KUKA KRL program: EPS_2_25369_MH3A_A_20251128065458.src

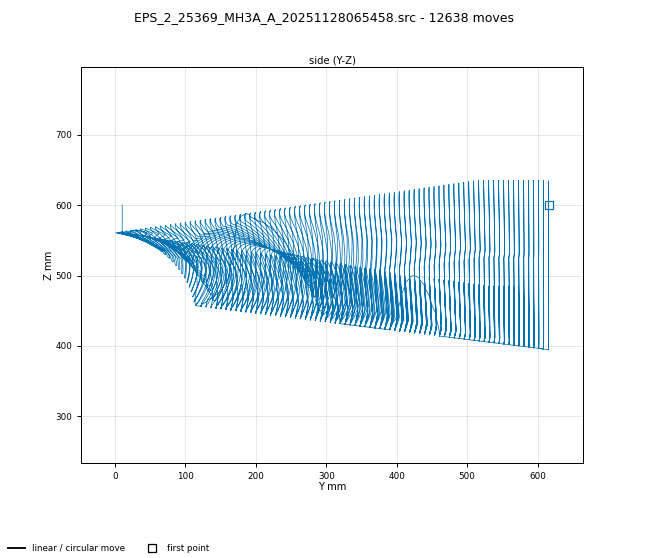
[picture p0: tool path of EPS_2_25369_MH3A_A_20251128065458.src, 12638 of 12640 moves have a stored position in this frame; points joined in program order, loops and branches not executed]
&ACCESS RVP
&REL 4
&COMMENT QRS 19112012
&PARAM EDITMASK = *
DEF PART()
EXT BAS (BAS_COMMAND :IN,REAL :IN )
INT I
BAS (#INITMOV,0 )

;KUKA QRS Post kuka4.cps  Date:22-06-2017 !

File_ID=2933

QRS_PRE_INIT()

;Init var - Until changes are made in qrs_pre_init
Outlet_Square_prg=0
Inlet_1_Square_prg=0
Inlet_2_Square_prg=0
Inlet_3_Square_prg=0
Inlet_4_Square_prg=0
Inlet_5_Square_prg=0

Outlet_1={X 0.000, Y 515.340, Z 534.500, B 0.000, E1 0.000 }
Inlet_1={X 0.000, Y 526.220, Z 384.500, B 0.000, E1 183.000 }
Inlet_2={X 0.000, Y 526.220, Z 384.500, B 0.000, E1 271.000 }
Outlet_1_type=201
Inlet_1_type=201
Inlet_2_type=201
;QRS#1=Sidecore dimensions
;QRS#2=200-8" PVC SDR 35
;QRS#3=200-8" PVC SDR 35
;QRS#4=200-8" PVC SDR 35
;QRS#5=
;QRS#6=
;QRS#7=
;QRS#8=
;QRS#9=12-08 PSX
;QRS#10=12-08 PSX
;QRS#11=12-08 PSX
;QRS#12=
;QRS#13=
;QRS#14=
;QRS#15=
;QRS#16=1220x127x914 3'
;QRS#17=EPS Height
;QRS#18=635
;QRS#19=*
;QRS#20= UPDATED VERSION 22-06-2017
;QRS#21=*
Outlet_Square=0100
Inlet_1_Square=0100
Inlet_2_Square=0100
Inlet_3_Square=0
Inlet_4_Square=0
Inlet_5_Square=0
Mill_Square=1
Outlet_Square_Prg=204
Inlet_1_Square_prg=204
Inlet_2_Square_prg=204

QRS_INIT()

$ADVANCE=5

; T1
PTP {E1 173.603,E2 173.603}
PTP {X 0,Y 615.513,A -85,B 0,C 180,E1 173.603,E2 173.603,E3 0,E4 0,E5 0,E6 0}
QRS_SPEED_INIT()
LIN {X 0,Y 615.513,Z 600,A -85,B 0,C 180,E1 173.603,E2 173.603,E3 0,E4 0,E5 0,E6 0} C_VEL
LIN {X 0,Y 615.513,Z 404.872,A -85,B 0,C 180,E1 173.603,E2 173.603} C_VEL
LIN {X 0,Y 615.513,Z 396.699,A -85,B 0,C 180,E1 173.603,E2 173.603} C_VEL
LIN {X 0,Y 615.495,Z 394.699,A -85,B 0,C 180,E1 173.416,E2 173.416} C_VEL
LIN {X 0,Y 615.488,Z 394.697,A -85,B 0,C 180,E1 170.801,E2 170.801} C_VEL
LIN {X 0,Y 615.484,Z 394.699,A -85,B 0,C 180,E1 168.139,E2 168.139} C_VEL
LIN {X 0,Y 615.49,Z 394.698,A -85,B 0,C 180,E1 165.451,E2 165.451} C_VEL
LIN {X 0,Y 615.49,Z 394.698,A -85,B 0,C 180,E1 162.729,E2 162.729} C_VEL
LIN {X 0,Y 615.486,Z 394.698,A -85,B 0,C 180,E1 159.967,E2 159.967} C_VEL
LIN {X 0,Y 615.489,Z 394.7,A -85,B 0,C 180,E1 157.155,E2 157.155} C_VEL
LIN {X 0,Y 615.486,Z 394.697,A -85,B 0,C 180,E1 154.432,E2 154.432} C_VEL
LIN {X 0,Y 615.493,Z 394.7,A -85,B 0,C 180,E1 151.549,E2 151.549} C_VEL
LIN {X 0,Y 615.483,Z 394.698,A -85,B 0,C 180,E1 148.915,E2 148.915} C_VEL
LIN {X 0,Y 615.486,Z 394.699,A -85,B 0,C 180,E1 146.466,E2 146.466} C_VEL
LIN {X 0,Y 615.491,Z 394.7,A -85,B 0,C 180,E1 144.166,E2 144.166} C_VEL
LIN {X 0,Y 615.493,Z 394.7,A -85,B 0,C 180,E1 141.931,E2 141.931} C_VEL
LIN {X 0,Y 615.48,Z 394.699,A -85,B 0,C 180,E1 139.393,E2 139.393} C_VEL
LIN {X 0,Y 615.498,Z 394.696,A -85,B 0,C 180,E1 136.756,E2 136.756} C_VEL
LIN {X 0,Y 615.493,Z 394.697,A -85,B 0,C 180,E1 133.998,E2 133.998} C_VEL
LIN {X 0,Y 615.49,Z 394.701,A -85,B 0,C 180,E1 131.094,E2 131.094} C_VEL
LIN {X 0,Y 615.493,Z 394.701,A -85,B 0,C 180,E1 128.904,E2 128.904} C_VEL
LIN {X 0,Y 615.483,Z 394.699,A -85,B 0,C 180,E1 126.425,E2 126.425} C_VEL
LIN {X 0,Y 615.488,Z 394.696,A -85,B 0,C 180,E1 124.022,E2 124.022} C_VEL
LIN {X 0,Y 615.493,Z 394.696,A -85,B 0,C 180,E1 121.685,E2 121.685} C_VEL
LIN {X 0,Y 615.488,Z 394.698,A -85,B 0,C 180,E1 119.406,E2 119.406} C_VEL
LIN {X 0,Y 615.491,Z 394.7,A -85,B 0,C 180,E1 117.045,E2 117.045} C_VEL
LIN {X 0,Y 615.479,Z 394.699,A -85,B 0,C 180,E1 114.272,E2 114.272} C_VEL
LIN {X 0,Y 615.49,Z 394.7,A -85,B 0,C 180,E1 111.432,E2 111.432} C_VEL
LIN {X 0,Y 615.482,Z 394.699,A -85,B 0,C 180,E1 108.602,E2 108.602} C_VEL
LIN {X 0,Y 615.492,Z 394.698,A -85,B 0,C 180,E1 105.905,E2 105.905} C_VEL
LIN {X 0,Y 615.48,Z 394.699,A -85,B 0,C 180,E1 103.201,E2 103.201} C_VEL
LIN {X 0,Y 615.487,Z 394.699,A -85,B 0,C 180,E1 100.527,E2 100.527} C_VEL
LIN {X 0,Y 615.492,Z 394.697,A -85,B 0,C 180,E1 98.247,E2 98.247} C_VEL
LIN {X 0,Y 615.49,Z 407.911,A -85,B 0,C 180,E1 97.793,E2 97.793} C_VEL
LIN {X 0,Y 615.49,Z 420.359,A -85,B 0,C 180,E1 97.216,E2 97.216} C_VEL
LIN {X 0,Y 615.488,Z 431.447,A -85,B 0,C 180,E1 96.557,E2 96.557} C_VEL
LIN {X 0,Y 615.498,Z 441.465,A -85,B 0,C 180,E1 95.816,E2 95.816} C_VEL
LIN {X 0,Y 615.498,Z 451.287,A -85,B 0,C 180,E1 94.913,E2 94.913} C_VEL
LIN {X 0,Y 615.497,Z 459.947,A -85,B 0,C 180,E1 93.928,E2 93.928} C_VEL
LIN {X 0,Y 615.497,Z 466.864,A -85,B 0,C 180,E1 92.945,E2 92.945} C_VEL
LIN {X 0,Y 615.5,Z 472.408,A -85,B 0,C 180,E1 91.963,E2 91.963} C_VEL
LIN {X 0,Y 615.497,Z 476.776,A -85,B 0,C 180,E1 90.981,E2 90.981} C_VEL
LIN {X 0,Y 615.496,Z 480.091,A -85,B 0,C 180,E1 90,E2 90} C_VEL
LIN {X 0,Y 615.498,Z 482.985,A -85,B 0,C 180,E1 88.691,E2 88.691} C_VEL
LIN {X 0,Y 615.499,Z 483.848,A -85,B 0,C 180,E1 88.037,E2 88.037} C_VEL
LIN {X 0,Y 615.496,Z 484.294,A -85,B 0,C 180,E1 87.382,E2 87.382} C_VEL
LIN {X 0,Y 615.495,Z 484.012,A -85,B 0,C 180,E1 86.071,E2 86.071} C_VEL
LIN {X 0,Y 615.495,Z 483.305,A -85,B 0,C 180,E1 85.415,E2 85.415} C_VEL
LIN {X 0,Y 615.496,Z 482.159,A -85,B 0,C 180,E1 84.759,E2 84.759} C_VEL
LIN {X 0,Y 615.497,Z 480.602,A -85,B 0,C 180,E1 84.101,E2 84.101} C_VEL
LIN {X 0,Y 615.497,Z 477.422,A -85,B 0,C 180,E1 83.102,E2 83.102} C_VEL
LIN {X 0,Y 615.495,Z 473.273,A -85,B 0,C 180,E1 82.124,E2 82.124} C_VEL
LIN {X 0,Y 615.496,Z 466.876,A -85,B 0,C 180,E1 80.967,E2 80.967} C_VEL
LIN {X 0,Y 615.497,Z 459.868,A -85,B 0,C 180,E1 79.972,E2 79.972} C_VEL
LIN {X 0,Y 615.498,Z 450.905,A -85,B 0,C 180,E1 78.958,E2 78.958} C_VEL
LIN {X 0,Y 615.497,Z 442.001,A -85,B 0,C 180,E1 78.139,E2 78.139} C_VEL
LIN {X 0,Y 615.484,Z 431.945,A -85,B 0,C 180,E1 77.386,E2 77.386} C_VEL
LIN {X 0,Y 615.477,Z 420.738,A -85,B 0,C 180,E1 76.714,E2 76.714} C_VEL
LIN {X 0,Y 615.487,Z 410.114,A -85,B 0,C 180,E1 76.21,E2 76.21} C_VEL
LIN {X 0,Y 615.492,Z 397.644,A -85,B 0,C 180,E1 75.758,E2 75.758} C_VEL
LIN {X 0,Y 615.493,Z 394.697,A -85,B 0,C 180,E1 75.662,E2 75.662} C_VEL
LIN {X 0,Y 615.487,Z 394.697,A -85,B 0,C 180,E1 73.413,E2 73.413} C_VEL
LIN {X 0,Y 615.475,Z 394.685,A -85,B 0,C 180,E1 70.661,E2 70.661} C_VEL
LIN {X 0,Y 615.493,Z 394.694,A -85,B 0,C 180,E1 67.864,E2 67.864} C_VEL
LIN {X 0,Y 615.488,Z 394.684,A -85,B 0,C 180,E1 65.008,E2 65.008} C_VEL
LIN {X 0,Y 615.48,Z 394.684,A -85,B 0,C 180,E1 62.822,E2 62.822} C_VEL
LIN {X 0,Y 615.497,Z 394.686,A -85,B 0,C 180,E1 60.205,E2 60.205} C_VEL
LIN {X 0,Y 615.479,Z 394.696,A -85,B 0,C 180,E1 57.542,E2 57.542} C_VEL
LIN {X 0,Y 615.499,Z 394.683,A -85,B 0,C 180,E1 55.185,E2 55.185} C_VEL
LIN {X 0,Y 615.477,Z 394.685,A -85,B 0,C 180,E1 52.757,E2 52.757} C_VEL
LIN {X 0,Y 615.498,Z 394.699,A -85,B 0,C 180,E1 49.91,E2 49.91} C_VEL
LIN {X 0,Y 615.481,Z 394.684,A -85,B 0,C 180,E1 46.954,E2 46.954} C_VEL
LIN {X 0,Y 615.49,Z 394.7,A -85,B 0,C 180,E1 43.997,E2 43.997} C_VEL
LIN {X 0,Y 615.485,Z 394.688,A -85,B 0,C 180,E1 41.474,E2 41.474} C_VEL
LIN {X 0,Y 615.478,Z 394.685,A -85,B 0,C 180,E1 38.905,E2 38.905} C_VEL
LIN {X 0,Y 615.488,Z 394.69,A -85,B 0,C 180,E1 36.425,E2 36.425} C_VEL
LIN {X 0,Y 615.484,Z 394.687,A -85,B 0,C 180,E1 33.533,E2 33.533} C_VEL
LIN {X 0,Y 615.478,Z 394.685,A -85,B 0,C 180,E1 30.921,E2 30.921} C_VEL
LIN {X 0,Y 615.491,Z 394.691,A -85,B 0,C 180,E1 28.45,E2 28.45} C_VEL
LIN {X 0,Y 615.486,Z 394.686,A -85,B 0,C 180,E1 25.568,E2 25.568} C_VEL
LIN {X 0,Y 615.475,Z 394.688,A -85,B 0,C 180,E1 22.845,E2 22.845} C_VEL
LIN {X 0,Y 615.487,Z 394.692,A -85,B 0,C 180,E1 20.556,E2 20.556} C_VEL
LIN {X 0,Y 615.482,Z 394.694,A -85,B 0,C 180,E1 17.957,E2 17.957} C_VEL
LIN {X 0,Y 615.486,Z 394.683,A -85,B 0,C 180,E1 15.226,E2 15.226} C_VEL
LIN {X 0,Y 615.486,Z 394.696,A -85,B 0,C 180,E1 12.53,E2 12.53} C_VEL
LIN {X 0,Y 615.483,Z 394.699,A -85,B 0,C 180,E1 10.236,E2 10.236} C_VEL
LIN {X 0,Y 615.478,Z 407.188,A -85,B 0,C 180,E1 9.821,E2 9.821} C_VEL
LIN {X 0,Y 615.486,Z 419.115,A -85,B 0,C 180,E1 9.282,E2 9.282} C_VEL
LIN {X 0,Y 615.487,Z 430.482,A -85,B 0,C 180,E1 8.619,E2 8.619} C_VEL
LIN {X 0,Y 615.498,Z 440.718,A -85,B 0,C 180,E1 7.876,E2 7.876} C_VEL
LIN {X 0,Y 615.499,Z 449.87,A -85,B 0,C 180,E1 7.057,E2 7.057} C_VEL
LIN {X 0,Y 615.496,Z 458.846,A -85,B 0,C 180,E1 6.063,E2 6.063} C_VEL
LIN {X 0,Y 615.497,Z 466.028,A -85,B 0,C 180,E1 5.077,E2 5.077} C_VEL
LIN {X 0,Y 615.496,Z 470.874,A -85,B 0,C 180,E1 4.257,E2 4.257} C_VEL
LIN {X 0,Y 615.496,Z 475.586,A -85,B 0,C 180,E1 3.273,E2 3.273} C_VEL
LIN {X 0,Y 615.498,Z 479.197,A -85,B 0,C 180,E1 2.291,E2 2.291} C_VEL
LIN {X 0,Y 615.496,Z 481.817,A -85,B 0,C 180,E1 1.309,E2 1.309} C_VEL
LIN {X 0,Y 615.495,Z 483.889,A -85,B 0,C 180,E1 0,E2 0} C_VEL
LIN {X 0,Y 615.496,Z 484.331,A -85,B 0,C 180,E1 -1.308,E2 -1.308} C_VEL
LIN {X 0,Y 615.495,Z 483.257,A -85,B 0,C 180,E1 -2.618,E2 -2.618} C_VEL
LIN {X 0,Y 615.497,Z 482.09,A -85,B 0,C 180,E1 -3.273,E2 -3.273} C_VEL
LIN {X 0,Y 615.494,Z 480.523,A -85,B 0,C 180,E1 -3.928,E2 -3.928} C_VEL
LIN {X 0,Y 615.494,Z 477.369,A -85,B 0,C 180,E1 -4.913,E2 -4.913} C_VEL
LIN {X 0,Y 615.498,Z 473.162,A -85,B 0,C 180,E1 -5.898,E2 -5.898} C_VEL
LIN {X 0,Y 615.497,Z 466.732,A -85,B 0,C 180,E1 -7.057,E2 -7.057} C_VEL
LIN {X 0,Y 615.498,Z 459.768,A -85,B 0,C 180,E1 -8.041,E2 -8.041} C_VEL
LIN {X 0,Y 615.497,Z 450.99,A -85,B 0,C 180,E1 -9.033,E2 -9.033} C_VEL
LIN {X 0,Y 615.499,Z 441.987,A -85,B 0,C 180,E1 -9.862,E2 -9.862} C_VEL
LIN {X 0,Y 615.488,Z 431.924,A -85,B 0,C 180,E1 -10.615,E2 -10.615} C_VEL
LIN {X 0,Y 615.488,Z 420.906,A -85,B 0,C 180,E1 -11.276,E2 -11.276} C_VEL
LIN {X 0,Y 615.487,Z 408.448,A -85,B 0,C 180,E1 -11.861,E2 -11.861} C_VEL
LIN {X 0,Y 615.489,Z 396.407,A -85,B 0,C 180,E1 -12.279,E2 -12.279} C_VEL
LIN {X 0,Y 615.488,Z 394.694,A -85,B 0,C 180,E1 -12.342,E2 -12.342} C_VEL
LIN {X 0,Y 615.49,Z 394.692,A -85,B 0,C 180,E1 -15.226,E2 -15.226} C_VEL
LIN {X 0,Y 615.477,Z 394.696,A -85,B 0,C 180,E1 -17.957,E2 -17.957} C_VEL
LIN {X 0,Y 615.477,Z 394.696,A -85,B 0,C 180,E1 -20.731,E2 -20.731} C_VEL
LIN {X 0,Y 615.486,Z 394.694,A -85,B 0,C 180,E1 -23.556,E2 -23.556} C_VEL
LIN {X 0,Y 615.493,Z 394.691,A -85,B 0,C 180,E1 -26.444,E2 -26.444} C_VEL
LIN {X 0,Y 615.492,Z 394.692,A -85,B 0,C 180,E1 -29.406,E2 -29.406} C_VEL
LIN {X 0,Y 615.492,Z 394.693,A -85,B 0,C 180,E1 -32.331,E2 -32.331} C_VEL
LIN {X 0,Y 615.477,Z 394.695,A -85,B 0,C 180,E1 -34.816,E2 -34.816} C_VEL
LIN {X 0,Y 615.494,Z 394.694,A -85,B 0,C 180,E1 -37.242,E2 -37.242} C_VEL
LIN {X 0,Y 615.488,Z 394.695,A -85,B 0,C 180,E1 -40.089,E2 -40.089} C_VEL
LIN {X 0,Y 615.499,Z 394.696,A -85,B 0,C 180,E1 -42.352,E2 -42.352} C_VEL
LIN {X 0,Y 615.48,Z 394.699,A -85,B 0,C 180,E1 -45.069,E2 -45.069} C_VEL
LIN {X 0,Y 615.487,Z 394.699,A -85,B 0,C 180,E1 -47.92,E2 -47.92} C_VEL
LIN {X 0,Y 615.494,Z 394.691,A -85,B 0,C 180,E1 -50.25,E2 -50.25} C_VEL
LIN {X 0,Y 615.482,Z 394.694,A -85,B 0,C 180,E1 -53.064,E2 -53.064} C_VEL
LIN {X 0,Y 615.479,Z 394.815,A -85,B 0,C 180,E1 -54.534,E2 -54.534} C_VEL
LIN {X 0,Y 615.489,Z 408.626,A -85,B 0,C 180,E1 -57.154,E2 -57.154} C_VEL
LIN {X 0,Y 615.476,Z 422.321,A -85,B 0,C 180,E1 -59.839,E2 -59.839} C_VEL
LIN {X 0,Y 615.481,Z 436.016,A -85,B 0,C 180,E1 -62.454,E2 -62.454} C_VEL
LIN {X 0,Y 615.497,Z 449.705,A -85,B 0,C 180,E1 -65.008,E2 -65.008} C_VEL
LIN {X 0,Y 615.487,Z 465.337,A -85,B 0,C 180,E1 -67.863,E2 -67.863} C_VEL
LIN {X 0,Y 615.492,Z 480.953,A -85,B 0,C 180,E1 -70.662,E2 -70.662} C_VEL
LIN {X 0,Y 615.492,Z 496.555,A -85,B 0,C 180,E1 -73.413,E2 -73.413} C_VEL
LIN {X 0,Y 615.498,Z 512.141,A -85,B 0,C 180,E1 -76.126,E2 -76.126} C_VEL
LIN {X 0,Y 615.482,Z 524.926,A -85,B 0,C 180,E1 -78.327,E2 -78.327} C_VEL
LIN {X 0,Y 615.477,Z 538.234,A -85,B 0,C 180,E1 -78.556,E2 -78.556} C_VEL
LIN {X 0,Y 615.489,Z 551.332,A -85,B 0,C 180,E1 -78.922,E2 -78.922} C_VEL
LIN {X 0,Y 615.48,Z 563.127,A -85,B 0,C 180,E1 -79.383,E2 -79.383} C_VEL
LIN {X 0,Y 615.486,Z 574.572,A -85,B 0,C 180,E1 -79.972,E2 -79.972} C_VEL
LIN {X 0,Y 615.499,Z 586.019,A -85,B 0,C 180,E1 -80.718,E2 -80.718} C_VEL
LIN {X 0,Y 615.498,Z 595.255,A -85,B 0,C 180,E1 -81.463,E2 -81.463} C_VEL
LIN {X 0,Y 615.499,Z 603.652,A -85,B 0,C 180,E1 -82.289,E2 -82.289} C_VEL
LIN {X 0,Y 615.497,Z 611.69,A -85,B 0,C 180,E1 -83.259,E2 -83.259} C_VEL
LIN {X 0,Y 615.498,Z 617.422,A -85,B 0,C 180,E1 -84.101,E2 -84.101} C_VEL
LIN {X 0,Y 615.497,Z 622.871,A -85,B 0,C 180,E1 -85.087,E2 -85.087} C_VEL
LIN {X 0,Y 615.496,Z 627.14,A -85,B 0,C 180,E1 -86.071,E2 -86.071} C_VEL
LIN {X 0,Y 615.495,Z 629.398,A -85,B 0,C 180,E1 -86.727,E2 -86.727} C_VEL
LIN {X 0,Y 615.497,Z 631.232,A -85,B 0,C 180,E1 -87.382,E2 -87.382} C_VEL
LIN {X 0,Y 615.497,Z 632.608,A -85,B 0,C 180,E1 -88.037,E2 -88.037} C_VEL
LIN {X 0,Y 615.496,Z 634.173,A -85,B 0,C 180,E1 -89.346,E2 -89.346} C_VEL
LIN {X 0,Y 615.494,Z 634.389,A -85,B 0,C 180,E1 -90,E2 -90} C_VEL
LIN {X 0,Y 615.496,Z 633.58,A -85,B 0,C 180,E1 -91.308,E2 -91.308} C_VEL
LIN {X 0,Y 615.497,Z 632.608,A -85,B 0,C 180,E1 -91.963,E2 -91.963} C_VEL
LIN {X 0,Y 615.497,Z 631.233,A -85,B 0,C 180,E1 -92.618,E2 -92.618} C_VEL
LIN {X 0,Y 615.496,Z 628.35,A -85,B 0,C 180,E1 -93.6,E2 -93.6} C_VEL
LIN {X 0,Y 615.498,Z 624.442,A -85,B 0,C 180,E1 -94.584,E2 -94.584} C_VEL
LIN {X 0,Y 615.499,Z 619.405,A -85,B 0,C 180,E1 -95.57,E2 -95.57} C_VEL
LIN {X 0,Y 615.497,Z 612.869,A -85,B 0,C 180,E1 -96.583,E2 -96.583} C_VEL
LIN {X 0,Y 615.497,Z 605.134,A -85,B 0,C 180,E1 -97.545,E2 -97.545} C_VEL
LIN {X 0,Y 615.498,Z 597.046,A -85,B 0,C 180,E1 -98.371,E2 -98.371} C_VEL
LIN {X 0,Y 615.499,Z 587.169,A -85,B 0,C 180,E1 -99.198,E2 -99.198} C_VEL
LIN {X 0,Y 615.488,Z 575.983,A -85,B 0,C 180,E1 -99.945,E2 -99.945} C_VEL
LIN {X 0,Y 615.478,Z 565.026,A -85,B 0,C 180,E1 -100.527,E2 -100.527} C_VEL
LIN {X 0,Y 615.489,Z 552.505,A -85,B 0,C 180,E1 -101.039,E2 -101.039} C_VEL
LIN {X 0,Y 615.477,Z 540.071,A -85,B 0,C 180,E1 -101.402,E2 -101.402} C_VEL
LIN {X 0,Y 615.481,Z 526.474,A -85,B 0,C 180,E1 -101.652,E2 -101.652} C_VEL
LIN {X 0,Y 615.483,Z 524.799,A -85,B 0,C 180,E1 -101.694,E2 -101.694} C_VEL
LIN {X 0,Y 615.48,Z 510.017,A -85,B 0,C 180,E1 -104.242,E2 -104.242} C_VEL
LIN {X 0,Y 615.494,Z 494.605,A -85,B 0,C 180,E1 -106.928,E2 -106.928} C_VEL
LIN {X 0,Y 615.495,Z 479.002,A -85,B 0,C 180,E1 -109.685,E2 -109.685} C_VEL
LIN {X 0,Y 615.494,Z 462.802,A -85,B 0,C 180,E1 -112.595,E2 -112.595} C_VEL
LIN {X 0,Y 615.485,Z 448.151,A -85,B 0,C 180,E1 -115.279,E2 -115.279} C_VEL
LIN {X 0,Y 615.493,Z 434.061,A -85,B 0,C 180,E1 -117.915,E2 -117.915} C_VEL
LIN {X 0,Y 615.478,Z 420.366,A -85,B 0,C 180,E1 -120.54,E2 -120.54} C_VEL
LIN {X 0,Y 615.491,Z 406.665,A -85,B 0,C 180,E1 -123.236,E2 -123.236} C_VEL
LIN {X 0,Y 615.482,Z 394.698,A -85,B 0,C 180,E1 -125.516,E2 -125.516} C_VEL
LIN {X 0,Y 615.493,Z 394.699,A -85,B 0,C 180,E1 -128.068,E2 -128.068} C_VEL
LIN {X 0,Y 615.493,Z 394.697,A -85,B 0,C 180,E1 -130.606,E2 -130.606} C_VEL
LIN {X 0,Y 615.481,Z 394.699,A -85,B 0,C 180,E1 -133.245,E2 -133.245} C_VEL
LIN {X 0,Y 615.485,Z 394.7,A -85,B 0,C 180,E1 -136.003,E2 -136.003} C_VEL
LIN {X 0,Y 615.496,Z 394.698,A -85,B 0,C 180,E1 -138.905,E2 -138.905} C_VEL
LIN {X 0,Y 615.493,Z 394.699,A -85,B 0,C 180,E1 -141.096,E2 -141.096} C_VEL
LIN {X 0,Y 615.495,Z 394.697,A -85,B 0,C 180,E1 -143.576,E2 -143.576} C_VEL
LIN {X 0,Y 615.486,Z 394.7,A -85,B 0,C 180,E1 -146.466,E2 -146.466} C_VEL
LIN {X 0,Y 615.481,Z 394.7,A -85,B 0,C 180,E1 -149.08,E2 -149.08} C_VEL
LIN {X 0,Y 615.492,Z 394.696,A -85,B 0,C 180,E1 -151.549,E2 -151.549} C_VEL
LIN {X 0,Y 615.496,Z 394.697,A -85,B 0,C 180,E1 -154.43,E2 -154.43} C_VEL
LIN {X 0,Y 615.485,Z 394.698,A -85,B 0,C 180,E1 -157.155,E2 -157.155} C_VEL
LIN {X 0,Y 615.487,Z 394.7,A -85,B 0,C 180,E1 -159.444,E2 -159.444} C_VEL
LIN {X 0,Y 615.483,Z 394.699,A -85,B 0,C 180,E1 -162.043,E2 -162.043} C_VEL
LIN {X 0,Y 615.495,Z 394.696,A -85,B 0,C 180,E1 -164.774,E2 -164.774} C_VEL
LIN {X 0,Y 615.493,Z 394.697,A -85,B 0,C 180,E1 -167.47,E2 -167.47} C_VEL
LIN {X 0,Y 615.479,Z 394.7,A -85,B 0,C 180,E1 -170.138,E2 -170.138} C_VEL
LIN {X 0,Y 615.484,Z 394.701,A -85,B 0,C 180,E1 -172.784,E2 -172.784} C_VEL
LIN {X 0,Y 615.492,Z 394.696,A -85,B 0,C 180,E1 -175.416,E2 -175.416} C_VEL
LIN {X 0,Y 615.5,Z 394.7,A -85,B 0,C 180,E1 -178.037,E2 -178.037} C_VEL
LIN {X 0,Y 615.489,Z 394.696,A -85,B 0,C 180,E1 -180.654,E2 -180.654} C_VEL
LIN {X 0,Y 615.486,Z 394.7,A -85,B 0,C 180,E1 -183.273,E2 -183.273} C_VEL
LIN {X 0,Y 615.482,Z 394.699,A -85,B 0,C 180,E1 -185.899,E2 -185.899} C_VEL
LIN {X 0,Y 615.495,Z 394.699,A -85,B 0,C 180,E1 -186.584,E2 -186.584} C_VEL
LIN {X 0,Y 614.812,Z 394.843,A -85,B 0,C 180,E1 -187.13,E2 -187.13} C_VEL
LIN {X 0,Y 611.974,Z 395.258,A -85,B 0,C 180,E1 -188.016,E2 -188.016} C_VEL
LIN {X 0,Y 609.584,Z 395.566,A -85,B 0,C 180,E1 -188.728,E2 -188.728} C_VEL
LIN {X 0,Y 608.551,Z 395.684,A -85,B 0,C 180,E1 -189.278,E2 -189.278} C_VEL
LIN {X 0,Y 608.462,Z 395.694,A -85,B 0,C 180,E1 -189.464,E2 -189.464} C_VEL
LIN {X 0,Y 608.462,Z 395.696,A -85,B 0,C 180,E1 -192,E2 -192} C_VEL
LIN {X 0,Y 608.478,Z 395.692,A -85,B 0,C 180,E1 -194.721,E2 -194.721} C_VEL
LIN {X 0,Y 608.454,Z 395.697,A -85,B 0,C 180,E1 -197.477,E2 -197.477} C_VEL
LIN {X 0,Y 608.467,Z 395.693,A -85,B 0,C 180,E1 -200.274,E2 -200.274} C_VEL
LIN {X 0,Y 608.461,Z 395.694,A -85,B 0,C 180,E1 -202.477,E2 -202.477} C_VEL
LIN {X 0,Y 608.461,Z 395.694,A -85,B 0,C 180,E1 -204.571,E2 -204.571} C_VEL
LIN {X 0,Y 608.48,Z 395.694,A -85,B 0,C 180,E1 -207.207,E2 -207.207} C_VEL
LIN {X 0,Y 608.466,Z 395.693,A -85,B 0,C 180,E1 -209.971,E2 -209.971} C_VEL
LIN {X 0,Y 608.463,Z 395.695,A -85,B 0,C 180,E1 -212.879,E2 -212.879} C_VEL
LIN {X 0,Y 608.444,Z 395.696,A -85,B 0,C 180,E1 -215.278,E2 -215.278} C_VEL
LIN {X 0,Y 608.473,Z 395.693,A -85,B 0,C 180,E1 -217.746,E2 -217.746} C_VEL
LIN {X 0,Y 608.448,Z 395.698,A -85,B 0,C 180,E1 -220.329,E2 -220.329} C_VEL
LIN {X 0,Y 608.485,Z 395.692,A -85,B 0,C 180,E1 -223.31,E2 -223.31} C_VEL
LIN {X 0,Y 608.478,Z 395.692,A -85,B 0,C 180,E1 -226.131,E2 -226.131} C_VEL
LIN {X 0,Y 608.459,Z 395.696,A -85,B 0,C 180,E1 -228.824,E2 -228.824} C_VEL
LIN {X 0,Y 608.472,Z 395.693,A -85,B 0,C 180,E1 -231.412,E2 -231.412} C_VEL
LIN {X 0,Y 608.465,Z 395.694,A -85,B 0,C 180,E1 -233.953,E2 -233.953} C_VEL
LIN {X 0,Y 608.472,Z 395.694,A -85,B 0,C 180,E1 -236.33,E2 -236.33} C_VEL
LIN {X 0,Y 608.483,Z 395.694,A -85,B 0,C 180,E1 -238.728,E2 -238.728} C_VEL
LIN {X 0,Y 608.471,Z 395.693,A -85,B 0,C 180,E1 -241.381,E2 -241.381} C_VEL
LIN {X 0,Y 608.443,Z 395.698,A -85,B 0,C 180,E1 -243.964,E2 -243.964} C_VEL
LIN {X 0,Y 608.468,Z 395.695,A -85,B 0,C 180,E1 -246.155,E2 -246.155} C_VEL
LIN {X 0,Y 608.471,Z 395.695,A -85,B 0,C 180,E1 -248.309,E2 -248.309} C_VEL
LIN {X 0,Y 608.457,Z 395.694,A -85,B 0,C 180,E1 -251.131,E2 -251.131} C_VEL
LIN {X 0,Y 608.463,Z 395.697,A -85,B 0,C 180,E1 -253.906,E2 -253.906} C_VEL
LIN {X 0,Y 608.462,Z 395.694,A -85,B 0,C 180,E1 -256.644,E2 -256.644} C_VEL
LIN {X 0,Y 608.467,Z 395.696,A -85,B 0,C 180,E1 -259.35,E2 -259.35} C_VEL
LIN {X 0,Y 608.464,Z 395.712,A -85,B 0,C 180,E1 -261.657,E2 -261.657} C_VEL
LIN {X 0,Y 608.521,Z 407.891,A -85,B 0,C 180,E1 -262.076,E2 -262.076} C_VEL
LIN {X 0,Y 608.507,Z 419.64,A -85,B 0,C 180,E1 -262.618,E2 -262.618} C_VEL
LIN {X 0,Y 608.48,Z 430.93,A -85,B 0,C 180,E1 -263.284,E2 -263.284} C_VEL
LIN {X 0,Y 608.498,Z 441.131,A -85,B 0,C 180,E1 -264.034,E2 -264.034} C_VEL
LIN {X 0,Y 608.483,Z 450.335,A -85,B 0,C 180,E1 -264.865,E2 -264.865} C_VEL
LIN {X 0,Y 608.474,Z 459.266,A -85,B 0,C 180,E1 -265.86,E2 -265.86} C_VEL
LIN {X 0,Y 608.459,Z 466.478,A -85,B 0,C 180,E1 -266.855,E2 -266.855} C_VEL
LIN {X 0,Y 608.46,Z 471.352,A -85,B 0,C 180,E1 -267.683,E2 -267.683} C_VEL
LIN {X 0,Y 608.449,Z 476.1,A -85,B 0,C 180,E1 -268.676,E2 -268.676} C_VEL
LIN {X 0,Y 608.441,Z 479.749,A -85,B 0,C 180,E1 -269.669,E2 -269.669} C_VEL
LIN {X 0,Y 608.437,Z 482.397,A -85,B 0,C 180,E1 -270.662,E2 -270.662} C_VEL
LIN {X 0,Y 608.45,Z 483.641,A -85,B 0,C 180,E1 -271.324,E2 -271.324} C_VEL
LIN {X 0,Y 608.444,Z 484.493,A -85,B 0,C 180,E1 -271.986,E2 -271.986} C_VEL
LIN {X 0,Y 608.422,Z 484.944,A -85,B 0,C 180,E1 -273.311,E2 -273.311} C_VEL
LIN {X 0,Y 608.432,Z 484.595,A -85,B 0,C 180,E1 -273.974,E2 -273.974} C_VEL
LIN {X 0,Y 608.428,Z 483.852,A -85,B 0,C 180,E1 -274.638,E2 -274.638} C_VEL
LIN {X 0,Y 608.438,Z 482.668,A -85,B 0,C 180,E1 -275.302,E2 -275.302} C_VEL
LIN {X 0,Y 608.448,Z 479.169,A -85,B 0,C 180,E1 -276.603,E2 -276.603} C_VEL
LIN {X 0,Y 608.449,Z 475.161,A -85,B 0,C 180,E1 -277.633,E2 -277.633} C_VEL
LIN {X 0,Y 608.451,Z 470.1,A -85,B 0,C 180,E1 -278.636,E2 -278.636} C_VEL
LIN {X 0,Y 608.467,Z 463.732,A -85,B 0,C 180,E1 -279.642,E2 -279.642} C_VEL
LIN {X 0,Y 608.451,Z 455.728,A -85,B 0,C 180,E1 -280.65,E2 -280.65} C_VEL
LIN {X 0,Y 608.471,Z 447.556,A -85,B 0,C 180,E1 -281.493,E2 -281.493} C_VEL
LIN {X 0,Y 608.477,Z 437.568,A -85,B 0,C 180,E1 -282.338,E2 -282.338} C_VEL
LIN {X 0,Y 608.498,Z 426.247,A -85,B 0,C 180,E1 -283.101,E2 -283.101} C_VEL
LIN {X 0,Y 608.503,Z 415.135,A -85,B 0,C 180,E1 -283.696,E2 -283.696} C_VEL
LIN {X 0,Y 608.533,Z 402.778,A -85,B 0,C 180,E1 -284.207,E2 -284.207} C_VEL
LIN {X 0,Y 608.466,Z 395.697,A -85,B 0,C 180,E1 -284.443,E2 -284.443} C_VEL
LIN {X 0,Y 608.446,Z 395.693,A -85,B 0,C 180,E1 -286.784,E2 -286.784} C_VEL
LIN {X 0,Y 608.449,Z 395.688,A -85,B 0,C 180,E1 -289.571,E2 -289.571} C_VEL
LIN {X 0,Y 608.465,Z 395.694,A -85,B 0,C 180,E1 -292.476,E2 -292.476} C_VEL
LIN {X 0,Y 608.457,Z 395.693,A -85,B 0,C 180,E1 -294.571,E2 -294.571} C_VEL
LIN {X 0,Y 608.477,Z 395.684,A -85,B 0,C 180,E1 -297.206,E2 -297.206} C_VEL
LIN {X 0,Y 608.477,Z 395.69,A -85,B 0,C 180,E1 -299.972,E2 -299.972} C_VEL
LIN {X 0,Y 608.452,Z 395.689,A -85,B 0,C 180,E1 -302.88,E2 -302.88} C_VEL
LIN {X 0,Y 608.447,Z 395.688,A -85,B 0,C 180,E1 -305.278,E2 -305.278} C_VEL
LIN {X 0,Y 608.477,Z 395.694,A -85,B 0,C 180,E1 -308.241,E2 -308.241} C_VEL
LIN {X 0,Y 608.457,Z 395.687,A -85,B 0,C 180,E1 -311.341,E2 -311.341} C_VEL
LIN {X 0,Y 608.459,Z 395.694,A -85,B 0,C 180,E1 -314.264,E2 -314.264} C_VEL
LIN {X 0,Y 608.453,Z 395.687,A -85,B 0,C 180,E1 -317.04,E2 -317.04} C_VEL
LIN {X 0,Y 608.458,Z 395.692,A -85,B 0,C 180,E1 -319.697,E2 -319.697} C_VEL
LIN {X 0,Y 608.472,Z 395.691,A -85,B 0,C 180,E1 -322.254,E2 -322.254} C_VEL
LIN {X 0,Y 608.444,Z 395.689,A -85,B 0,C 180,E1 -325.096,E2 -325.096} C_VEL
LIN {X 0,Y 608.461,Z 395.69,A -85,B 0,C 180,E1 -327.478,E2 -327.478} C_VEL
LIN {X 0,Y 608.463,Z 395.691,A -85,B 0,C 180,E1 -330.22,E2 -330.22} C_VEL
LIN {X 0,Y 608.478,Z 395.684,A -85,B 0,C 180,E1 -332.794,E2 -332.794} C_VEL
LIN {X 0,Y 608.454,Z 395.691,A -85,B 0,C 180,E1 -335.429,E2 -335.429} C_VEL
LIN {X 0,Y 608.472,Z 395.687,A -85,B 0,C 180,E1 -338.308,E2 -338.308} C_VEL
LIN {X 0,Y 608.472,Z 395.688,A -85,B 0,C 180,E1 -341.285,E2 -341.285} C_VEL
LIN {X 0,Y 608.458,Z 395.694,A -85,B 0,C 180,E1 -343.906,E2 -343.906} C_VEL
LIN {X 0,Y 608.461,Z 395.686,A -85,B 0,C 180,E1 -346.643,E2 -346.643} C_VEL
LIN {X 0,Y 608.477,Z 395.695,A -85,B 0,C 180,E1 -349.645,E2 -349.645} C_VEL
LIN {X 0,Y 608.51,Z 408.661,A -85,B 0,C 180,E1 -350.107,E2 -350.107} C_VEL
LIN {X 0,Y 608.503,Z 421.068,A -85,B 0,C 180,E1 -350.695,E2 -350.695} C_VEL
LIN {X 0,Y 608.501,Z 432.147,A -85,B 0,C 180,E1 -351.364,E2 -351.364} C_VEL
LIN {X 0,Y 608.494,Z 441.129,A -85,B 0,C 180,E1 -352.033,E2 -352.033} C_VEL
LIN {X 0,Y 608.467,Z 450.36,A -85,B 0,C 180,E1 -352.867,E2 -352.867} C_VEL
LIN {X 0,Y 608.446,Z 459.315,A -85,B 0,C 180,E1 -353.866,E2 -353.866} C_VEL
LIN {X 0,Y 608.446,Z 466.538,A -85,B 0,C 180,E1 -354.864,E2 -354.864} C_VEL
LIN {X 0,Y 608.441,Z 471.413,A -85,B 0,C 180,E1 -355.694,E2 -355.694} C_VEL
LIN {X 0,Y 608.43,Z 476.157,A -85,B 0,C 180,E1 -356.689,E2 -356.689} C_VEL
LIN {X 0,Y 608.43,Z 479.793,A -85,B 0,C 180,E1 -357.683,E2 -357.683} C_VEL
LIN {X 0,Y 608.448,Z 482.428,A -85,B 0,C 180,E1 -358.676,E2 -358.676} C_VEL
LIN {X 0,Y 608.436,Z 484.505,A -85,B 0,C 180,E1 -360,E2 -360} C_VEL
LIN {X 0,Y 608.448,Z 484.941,A -85,B 0,C 180,E1 -361.324,E2 -361.324} C_VEL
LIN {X 0,Y 608.442,Z 484.587,A -85,B 0,C 180,E1 -361.986,E2 -361.986} C_VEL
LIN {X 0,Y 608.422,Z 483.836,A -85,B 0,C 180,E1 -362.648,E2 -362.648} C_VEL
LIN {X 0,Y 608.425,Z 482.651,A -85,B 0,C 180,E1 -363.311,E2 -363.311} C_VEL
LIN {X 0,Y 608.432,Z 480.116,A -85,B 0,C 180,E1 -364.306,E2 -364.306} C_VEL
LIN {X 0,Y 608.441,Z 476.58,A -85,B 0,C 180,E1 -365.302,E2 -365.302} C_VEL
LIN {X 0,Y 608.452,Z 471.56,A -85,B 0,C 180,E1 -366.369,E2 -366.369} C_VEL
LIN {X 0,Y 608.451,Z 464.92,A -85,B 0,C 180,E1 -367.466,E2 -367.466} C_VEL
LIN {X 0,Y 608.464,Z 457.315,A -85,B 0,C 180,E1 -368.469,E2 -368.469} C_VEL
LIN {X 0,Y 608.46,Z 449.539,A -85,B 0,C 180,E1 -369.306,E2 -369.306} C_VEL
LIN {X 0,Y 608.491,Z 438.955,A -85,B 0,C 180,E1 -370.229,E2 -370.229} C_VEL
LIN {X 0,Y 608.494,Z 428.487,A -85,B 0,C 180,E1 -370.966,E2 -370.966} C_VEL
LIN {X 0,Y 608.506,Z 417.621,A -85,B 0,C 180,E1 -371.576,E2 -371.576} C_VEL
LIN {X 0,Y 608.519,Z 404.962,A -85,B 0,C 180,E1 -372.125,E2 -372.125} C_VEL
LIN {X 0,Y 608.471,Z 395.691,A -85,B 0,C 180,E1 -372.444,E2 -372.444} C_VEL
LIN {X 0,Y 608.476,Z 395.69,A -85,B 0,C 180,E1 -375.406,E2 -375.406} C_VEL
LIN {X 0,Y 608.443,Z 395.694,A -85,B 0,C 180,E1 -378.172,E2 -378.172} C_VEL
LIN {X 0,Y 608.457,Z 395.693,A -85,B 0,C 180,E1 -380.982,E2 -380.982} C_VEL
LIN {X 0,Y 608.449,Z 395.697,A -85,B 0,C 180,E1 -383.124,E2 -383.124} C_VEL
LIN {X 0,Y 608.481,Z 395.694,A -85,B 0,C 180,E1 -385.722,E2 -385.722} C_VEL
LIN {X 0,Y 608.48,Z 395.694,A -85,B 0,C 180,E1 -388.62,E2 -388.62} C_VEL
LIN {X 0,Y 608.448,Z 395.698,A -85,B 0,C 180,E1 -391.318,E2 -391.318} C_VEL
LIN {X 0,Y 608.475,Z 395.691,A -85,B 0,C 180,E1 -393.735,E2 -393.735} C_VEL
LIN {X 0,Y 608.449,Z 395.694,A -85,B 0,C 180,E1 -396.092,E2 -396.092} C_VEL
LIN {X 0,Y 608.436,Z 395.697,A -85,B 0,C 180,E1 -398.591,E2 -398.591} C_VEL
LIN {X 0,Y 608.462,Z 395.694,A -85,B 0,C 180,E1 -401.342,E2 -401.342} C_VEL
LIN {X 0,Y 608.464,Z 395.693,A -85,B 0,C 180,E1 -404.264,E2 -404.264} C_VEL
LIN {X 0,Y 608.455,Z 395.694,A -85,B 0,C 180,E1 -407.04,E2 -407.04} C_VEL
LIN {X 0,Y 608.456,Z 395.695,A -85,B 0,C 180,E1 -409.697,E2 -409.697} C_VEL
LIN {X 0,Y 608.467,Z 395.697,A -85,B 0,C 180,E1 -412.253,E2 -412.253} C_VEL
LIN {X 0,Y 608.485,Z 395.82,A -85,B 0,C 180,E1 -414.369,E2 -414.369} C_VEL
LIN {X 0,Y 608.571,Z 407.184,A -85,B 0,C 180,E1 -416.534,E2 -416.534} C_VEL
LIN {X 0,Y 608.636,Z 416.451,A -85,B 0,C 180,E1 -418.305,E2 -418.305} C_VEL
LIN {X 0,Y 608.599,Z 430.146,A -85,B 0,C 180,E1 -420.987,E2 -420.987} C_VEL
LIN {X 0,Y 608.552,Z 443.841,A -85,B 0,C 180,E1 -423.6,E2 -423.6} C_VEL
LIN {X 0,Y 608.532,Z 457.536,A -85,B 0,C 180,E1 -426.158,E2 -426.158} C_VEL
LIN {X 0,Y 608.522,Z 471.231,A -85,B 0,C 180,E1 -428.666,E2 -428.666} C_VEL
LIN {X 0,Y 608.494,Z 485.749,A -85,B 0,C 180,E1 -431.278,E2 -431.278} C_VEL
LIN {X 0,Y 608.483,Z 500.578,A -85,B 0,C 180,E1 -433.907,E2 -433.907} C_VEL
LIN {X 0,Y 608.464,Z 516.229,A -85,B 0,C 180,E1 -436.643,E2 -436.643} C_VEL
LIN {X 0,Y 608.447,Z 525.155,A -85,B 0,C 180,E1 -438.19,E2 -438.19} C_VEL
LIN {X 0,Y 608.537,Z 539.259,A -85,B 0,C 180,E1 -438.445,E2 -438.445} C_VEL
LIN {X 0,Y 608.524,Z 551.919,A -85,B 0,C 180,E1 -438.809,E2 -438.809} C_VEL
LIN {X 0,Y 608.507,Z 563.629,A -85,B 0,C 180,E1 -439.277,E2 -439.277} C_VEL
LIN {X 0,Y 608.494,Z 574.752,A -85,B 0,C 180,E1 -439.855,E2 -439.855} C_VEL
LIN {X 0,Y 608.504,Z 586.249,A -85,B 0,C 180,E1 -440.611,E2 -440.611} C_VEL
LIN {X 0,Y 608.472,Z 595.534,A -85,B 0,C 180,E1 -441.364,E2 -441.364} C_VEL
LIN {X 0,Y 608.456,Z 603.987,A -85,B 0,C 180,E1 -442.2,E2 -442.2} C_VEL
LIN {X 0,Y 608.462,Z 612.234,A -85,B 0,C 180,E1 -443.201,E2 -443.201} C_VEL
LIN {X 0,Y 608.437,Z 618.875,A -85,B 0,C 180,E1 -444.199,E2 -444.199} C_VEL
LIN {X 0,Y 608.432,Z 624.949,A -85,B 0,C 180,E1 -445.362,E2 -445.362} C_VEL
LIN {X 0,Y 608.449,Z 628.896,A -85,B 0,C 180,E1 -446.357,E2 -446.357} C_VEL
LIN {X 0,Y 608.425,Z 631.809,A -85,B 0,C 180,E1 -447.352,E2 -447.352} C_VEL
LIN {X 0,Y 608.442,Z 633.201,A -85,B 0,C 180,E1 -448.014,E2 -448.014} C_VEL
LIN {X 0,Y 608.438,Z 634.783,A -85,B 0,C 180,E1 -449.338,E2 -449.338} C_VEL
LIN {X 0,Y 608.434,Z 635,A -85,B 0,C 180,E1 -450,E2 -450} C_VEL
LIN {X 0,Y 608.448,Z 634.184,A -85,B 0,C 180,E1 -451.324,E2 -451.324} C_VEL
LIN {X 0,Y 608.443,Z 633.202,A -85,B 0,C 180,E1 -451.986,E2 -451.986} C_VEL
LIN {X 0,Y 608.425,Z 631.809,A -85,B 0,C 180,E1 -452.648,E2 -452.648} C_VEL
LIN {X 0,Y 608.449,Z 628.897,A -85,B 0,C 180,E1 -453.642,E2 -453.642} C_VEL
LIN {X 0,Y 608.432,Z 624.951,A -85,B 0,C 180,E1 -454.638,E2 -454.638} C_VEL
LIN {X 0,Y 608.437,Z 618.877,A -85,B 0,C 180,E1 -455.801,E2 -455.801} C_VEL
LIN {X 0,Y 608.462,Z 612.236,A -85,B 0,C 180,E1 -456.799,E2 -456.799} C_VEL
LIN {X 0,Y 608.456,Z 603.99,A -85,B 0,C 180,E1 -457.8,E2 -457.8} C_VEL
LIN {X 0,Y 608.472,Z 595.537,A -85,B 0,C 180,E1 -458.636,E2 -458.636} C_VEL
LIN {X 0,Y 608.48,Z 585.092,A -85,B 0,C 180,E1 -459.473,E2 -459.473} C_VEL
LIN {X 0,Y 608.494,Z 574.757,A -85,B 0,C 180,E1 -460.145,E2 -460.145} C_VEL
LIN {X 0,Y 608.51,Z 563.274,A -85,B 0,C 180,E1 -460.74,E2 -460.74} C_VEL
LIN {X 0,Y 608.53,Z 550.914,A -85,B 0,C 180,E1 -461.224,E2 -461.224} C_VEL
LIN {X 0,Y 608.537,Z 537.443,A -85,B 0,C 180,E1 -461.597,E2 -461.597} C_VEL
LIN {X 0,Y 608.447,Z 525.157,A -85,B 0,C 180,E1 -461.81,E2 -461.81} C_VEL
LIN {X 0,Y 608.479,Z 508.405,A -85,B 0,C 180,E1 -464.72,E2 -464.72} C_VEL
LIN {X 0,Y 608.492,Z 492.754,A -85,B 0,C 180,E1 -467.475,E2 -467.475} C_VEL
LIN {X 0,Y 608.516,Z 479.059,A -85,B 0,C 180,E1 -469.92,E2 -469.92} C_VEL
LIN {X 0,Y 608.549,Z 463.409,A -85,B 0,C 180,E1 -472.76,E2 -472.76} C_VEL
LIN {X 0,Y 608.563,Z 447.352,A -85,B 0,C 180,E1 -475.738,E2 -475.738} C_VEL
LIN {X 0,Y 608.608,Z 434.061,A -85,B 0,C 180,E1 -478.259,E2 -478.259} C_VEL
LIN {X 0,Y 608.614,Z 420.405,A -85,B 0,C 180,E1 -480.914,E2 -480.914} C_VEL
LIN {X 0,Y 608.61,Z 410.321,A -85,B 0,C 180,E1 -482.87,E2 -482.87} C_VEL
LIN {X 0,Y 608.595,Z 396.627,A -85,B 0,C 180,E1 -485.47,E2 -485.47} C_VEL
LIN {X 0,Y 608.479,Z 395.693,A -85,B 0,C 180,E1 -485.682,E2 -485.682} C_VEL
LIN {X 0,Y 608.474,Z 395.695,A -85,B 0,C 180,E1 -488.241,E2 -488.241} C_VEL
LIN {X 0,Y 608.452,Z 395.698,A -85,B 0,C 180,E1 -490.329,E2 -490.329} C_VEL
LIN {X 0,Y 608.47,Z 395.694,A -85,B 0,C 180,E1 -493.309,E2 -493.309} C_VEL
LIN {X 0,Y 608.472,Z 395.693,A -85,B 0,C 180,E1 -496.131,E2 -496.131} C_VEL
LIN {X 0,Y 608.464,Z 395.695,A -85,B 0,C 180,E1 -498.824,E2 -498.824} C_VEL
LIN {X 0,Y 608.474,Z 395.694,A -85,B 0,C 180,E1 -501.412,E2 -501.412} C_VEL
LIN {X 0,Y 608.462,Z 395.694,A -85,B 0,C 180,E1 -503.953,E2 -503.953} C_VEL
LIN {X 0,Y 608.451,Z 395.696,A -85,B 0,C 180,E1 -506.328,E2 -506.328} C_VEL
LIN {X 0,Y 608.448,Z 395.698,A -85,B 0,C 180,E1 -508.732,E2 -508.732} C_VEL
LIN {X 0,Y 608.475,Z 395.692,A -85,B 0,C 180,E1 -511.38,E2 -511.38} C_VEL
LIN {X 0,Y 608.455,Z 395.696,A -85,B 0,C 180,E1 -513.965,E2 -513.965} C_VEL
LIN {X 0,Y 608.468,Z 395.694,A -85,B 0,C 180,E1 -516.155,E2 -516.155} C_VEL
LIN {X 0,Y 608.474,Z 395.693,A -85,B 0,C 180,E1 -518.309,E2 -518.309} C_VEL
LIN {X 0,Y 608.471,Z 395.693,A -85,B 0,C 180,E1 -521.284,E2 -521.284} C_VEL
LIN {X 0,Y 608.468,Z 395.696,A -85,B 0,C 180,E1 -523.906,E2 -523.906} C_VEL
LIN {X 0,Y 608.47,Z 395.693,A -85,B 0,C 180,E1 -526.644,E2 -526.644} C_VEL
LIN {X 0,Y 608.471,Z 395.696,A -85,B 0,C 180,E1 -529.35,E2 -529.35} C_VEL
LIN {X 0,Y 608.471,Z 395.693,A -85,B 0,C 180,E1 -532.033,E2 -532.033} C_VEL
LIN {X 0,Y 608.474,Z 395.695,A -85,B 0,C 180,E1 -534.698,E2 -534.698} C_VEL
LIN {X 0,Y 608.482,Z 395.692,A -85,B 0,C 180,E1 -537.352,E2 -537.352} C_VEL
LIN {X 0,Y 608.476,Z 395.693,A -85,B 0,C 180,E1 -540,E2 -540} C_VEL
LIN {X 0,Y 608.481,Z 395.692,A -85,B 0,C 180,E1 -542.648,E2 -542.648} C_VEL
LIN {X 0,Y 608.464,Z 395.694,A -85,B 0,C 180,E1 -545.302,E2 -545.302} C_VEL
LIN {X 0,Y 608.482,Z 395.693,A -85,B 0,C 180,E1 -547.967,E2 -547.967} C_VEL
LIN {X 0,Y 608.462,Z 395.694,A -85,B 0,C 180,E1 -549.464,E2 -549.464} C_VEL
LIN {X 0,Y 607.783,Z 395.781,A -85,B 0,C 180,E1 -550.017,E2 -550.017} C_VEL
LIN {X 0,Y 604.927,Z 396.138,A -85,B 0,C 180,E1 -550.913,E2 -550.913} C_VEL
LIN {X 0,Y 602.524,Z 396.437,A -85,B 0,C 180,E1 -551.635,E2 -551.635} C_VEL
LIN {X 0,Y 601.495,Z 396.564,A -85,B 0,C 180,E1 -552.192,E2 -552.192} C_VEL
LIN {X 0,Y 601.412,Z 396.573,A -85,B 0,C 180,E1 -552.38,E2 -552.38} C_VEL
LIN {X 0,Y 601.432,Z 396.57,A -85,B 0,C 180,E1 -554.897,E2 -554.897} C_VEL
LIN {X 0,Y 601.434,Z 396.569,A -85,B 0,C 180,E1 -556.986,E2 -556.986} C_VEL
LIN {X 0,Y 601.41,Z 396.575,A -85,B 0,C 180,E1 -559.81,E2 -559.81} C_VEL
LIN {X 0,Y 601.418,Z 396.572,A -85,B 0,C 180,E1 -562.606,E2 -562.606} C_VEL
LIN {X 0,Y 601.408,Z 396.574,A -85,B 0,C 180,E1 -564.879,E2 -564.879} C_VEL
LIN {X 0,Y 601.416,Z 396.574,A -85,B 0,C 180,E1 -567.362,E2 -567.362} C_VEL
LIN {X 0,Y 601.43,Z 396.57,A -85,B 0,C 180,E1 -570.164,E2 -570.164} C_VEL
LIN {X 0,Y 601.429,Z 396.573,A -85,B 0,C 180,E1 -572.716,E2 -572.716} C_VEL
LIN {X 0,Y 601.403,Z 396.574,A -85,B 0,C 180,E1 -575.113,E2 -575.113} C_VEL
LIN {X 0,Y 601.439,Z 396.569,A -85,B 0,C 180,E1 -577.419,E2 -577.419} C_VEL
LIN {X 0,Y 601.404,Z 396.574,A -85,B 0,C 180,E1 -579.996,E2 -579.996} C_VEL
LIN {X 0,Y 601.416,Z 396.573,A -85,B 0,C 180,E1 -582.67,E2 -582.67} C_VEL
LIN {X 0,Y 601.43,Z 396.571,A -85,B 0,C 180,E1 -585.482,E2 -585.482} C_VEL
LIN {X 0,Y 601.43,Z 396.57,A -85,B 0,C 180,E1 -588.407,E2 -588.407} C_VEL
LIN {X 0,Y 601.439,Z 396.57,A -85,B 0,C 180,E1 -590.876,E2 -590.876} C_VEL
LIN {X 0,Y 601.411,Z 396.572,A -85,B 0,C 180,E1 -593.739,E2 -593.739} C_VEL
LIN {X 0,Y 601.44,Z 396.569,A -85,B 0,C 180,E1 -596.064,E2 -596.064} C_VEL
LIN {X 0,Y 601.447,Z 396.569,A -85,B 0,C 180,E1 -598.542,E2 -598.542} C_VEL
LIN {X 0,Y 601.431,Z 396.57,A -85,B 0,C 180,E1 -601.373,E2 -601.373} C_VEL
LIN {X 0,Y 601.402,Z 396.573,A -85,B 0,C 180,E1 -603.636,E2 -603.636} C_VEL
LIN {X 0,Y 601.424,Z 396.571,A -85,B 0,C 180,E1 -606.59,E2 -606.59} C_VEL
LIN {X 0,Y 601.438,Z 396.571,A -85,B 0,C 180,E1 -609.479,E2 -609.479} C_VEL
LIN {X 0,Y 601.406,Z 396.573,A -85,B 0,C 180,E1 -612.312,E2 -612.312} C_VEL
LIN {X 0,Y 601.418,Z 396.571,A -85,B 0,C 180,E1 -614.409,E2 -614.409} C_VEL
LIN {X 0,Y 601.416,Z 396.574,A -85,B 0,C 180,E1 -617.172,E2 -617.172} C_VEL
LIN {X 0,Y 601.441,Z 396.569,A -85,B 0,C 180,E1 -619.905,E2 -619.905} C_VEL
LIN {X 0,Y 601.459,Z 396.569,A -85,B 0,C 180,E1 -621.538,E2 -621.538} C_VEL
LIN {X 0,Y 601.536,Z 409.742,A -85,B 0,C 180,E1 -622.025,E2 -622.025} C_VEL
LIN {X 0,Y 601.493,Z 421.868,A -85,B 0,C 180,E1 -622.616,E2 -622.616} C_VEL
LIN {X 0,Y 601.464,Z 433.211,A -85,B 0,C 180,E1 -623.323,E2 -623.323} C_VEL
LIN {X 0,Y 601.428,Z 443.525,A -85,B 0,C 180,E1 -624.131,E2 -624.131} C_VEL
LIN {X 0,Y 601.419,Z 452.299,A -85,B 0,C 180,E1 -624.972,E2 -624.972} C_VEL
LIN {X 0,Y 601.394,Z 460.871,A -85,B 0,C 180,E1 -625.979,E2 -625.979} C_VEL
LIN {X 0,Y 601.384,Z 467.737,A -85,B 0,C 180,E1 -626.986,E2 -626.986} C_VEL
LIN {X 0,Y 601.351,Z 473.245,A -85,B 0,C 180,E1 -627.991,E2 -627.991} C_VEL
LIN {X 0,Y 601.337,Z 477.575,A -85,B 0,C 180,E1 -628.996,E2 -628.996} C_VEL
LIN {X 0,Y 601.337,Z 480.849,A -85,B 0,C 180,E1 -630,E2 -630} C_VEL
LIN {X 0,Y 601.35,Z 483.701,A -85,B 0,C 180,E1 -631.34,E2 -631.34} C_VEL
LIN {X 0,Y 601.343,Z 484.526,A -85,B 0,C 180,E1 -632.009,E2 -632.009} C_VEL
LIN {X 0,Y 601.338,Z 484.936,A -85,B 0,C 180,E1 -633.35,E2 -633.35} C_VEL
LIN {X 0,Y 601.342,Z 484.571,A -85,B 0,C 180,E1 -634.021,E2 -634.021} C_VEL
LIN {X 0,Y 601.327,Z 483.794,A -85,B 0,C 180,E1 -634.693,E2 -634.693} C_VEL
LIN {X 0,Y 601.349,Z 482.589,A -85,B 0,C 180,E1 -635.365,E2 -635.365} C_VEL
LIN {X 0,Y 601.349,Z 479.366,A -85,B 0,C 180,E1 -636.583,E2 -636.583} C_VEL
LIN {X 0,Y 601.354,Z 475.01,A -85,B 0,C 180,E1 -637.724,E2 -637.724} C_VEL
LIN {X 0,Y 601.361,Z 468.916,A -85,B 0,C 180,E1 -638.908,E2 -638.908} C_VEL
LIN {X 0,Y 601.389,Z 462.227,A -85,B 0,C 180,E1 -639.926,E2 -639.926} C_VEL
LIN {X 0,Y 601.402,Z 455.406,A -85,B 0,C 180,E1 -640.777,E2 -640.777} C_VEL
LIN {X 0,Y 601.434,Z 447.171,A -85,B 0,C 180,E1 -641.629,E2 -641.629} C_VEL
LIN {X 0,Y 601.46,Z 437.08,A -85,B 0,C 180,E1 -642.484,E2 -642.484} C_VEL
LIN {X 0,Y 601.477,Z 425.634,A -85,B 0,C 180,E1 -643.257,E2 -643.257} C_VEL
LIN {X 0,Y 601.523,Z 414.464,A -85,B 0,C 180,E1 -643.854,E2 -643.854} C_VEL
LIN {X 0,Y 601.577,Z 402.944,A -85,B 0,C 180,E1 -644.331,E2 -644.331} C_VEL
LIN {X 0,Y 601.447,Z 396.57,A -85,B 0,C 180,E1 -644.551,E2 -644.551} C_VEL
LIN {X 0,Y 601.418,Z 396.566,A -85,B 0,C 180,E1 -646.987,E2 -646.987} C_VEL
LIN {X 0,Y 601.406,Z 396.567,A -85,B 0,C 180,E1 -649.81,E2 -649.81} C_VEL
LIN {X 0,Y 601.417,Z 396.569,A -85,B 0,C 180,E1 -652.683,E2 -652.683} C_VEL
LIN {X 0,Y 601.405,Z 396.567,A -85,B 0,C 180,E1 -654.879,E2 -654.879} C_VEL
LIN {X 0,Y 601.416,Z 396.564,A -85,B 0,C 180,E1 -657.362,E2 -657.362} C_VEL
LIN {X 0,Y 601.435,Z 396.571,A -85,B 0,C 180,E1 -660.164,E2 -660.164} C_VEL
LIN {X 0,Y 601.418,Z 396.566,A -85,B 0,C 180,E1 -662.714,E2 -662.714} C_VEL
LIN {X 0,Y 601.418,Z 396.564,A -85,B 0,C 180,E1 -665.114,E2 -665.114} C_VEL
LIN {X 0,Y 601.439,Z 396.562,A -85,B 0,C 180,E1 -667.419,E2 -667.419} C_VEL
LIN {X 0,Y 601.408,Z 396.573,A -85,B 0,C 180,E1 -669.996,E2 -669.996} C_VEL
LIN {X 0,Y 601.411,Z 396.566,A -85,B 0,C 180,E1 -672.671,E2 -672.671} C_VEL
LIN {X 0,Y 601.432,Z 396.564,A -85,B 0,C 180,E1 -675.482,E2 -675.482} C_VEL
LIN {X 0,Y 601.427,Z 396.567,A -85,B 0,C 180,E1 -678.407,E2 -678.407} C_VEL
LIN {X 0,Y 601.435,Z 396.565,A -85,B 0,C 180,E1 -681.529,E2 -681.529} C_VEL
LIN {X 0,Y 601.389,Z 396.573,A -85,B 0,C 180,E1 -684.245,E2 -684.245} C_VEL
LIN {X 0,Y 601.423,Z 396.564,A -85,B 0,C 180,E1 -686.686,E2 -686.686} C_VEL
LIN {X 0,Y 601.417,Z 396.564,A -85,B 0,C 180,E1 -689.058,E2 -689.058} C_VEL
LIN {X 0,Y 601.433,Z 396.565,A -85,B 0,C 180,E1 -691.373,E2 -691.373} C_VEL
LIN {X 0,Y 601.404,Z 396.572,A -85,B 0,C 180,E1 -693.636,E2 -693.636} C_VEL
LIN {X 0,Y 601.456,Z 396.569,A -85,B 0,C 180,E1 -695.859,E2 -695.859} C_VEL
LIN {X 0,Y 601.41,Z 396.565,A -85,B 0,C 180,E1 -698.761,E2 -698.761} C_VEL
LIN {X 0,Y 601.42,Z 396.572,A -85,B 0,C 180,E1 -701.608,E2 -701.608} C_VEL
LIN {X 0,Y 601.413,Z 396.565,A -85,B 0,C 180,E1 -704.408,E2 -704.408} C_VEL
LIN {X 0,Y 601.42,Z 396.566,A -85,B 0,C 180,E1 -707.172,E2 -707.172} C_VEL
LIN {X 0,Y 601.424,Z 396.572,A -85,B 0,C 180,E1 -709.543,E2 -709.543} C_VEL
LIN {X 0,Y 601.547,Z 408.94,A -85,B 0,C 180,E1 -709.992,E2 -709.992} C_VEL
LIN {X 0,Y 601.494,Z 421.299,A -85,B 0,C 180,E1 -710.585,E2 -710.585} C_VEL
LIN {X 0,Y 601.485,Z 432.338,A -85,B 0,C 180,E1 -711.263,E2 -711.263} C_VEL
LIN {X 0,Y 601.453,Z 441.287,A -85,B 0,C 180,E1 -711.939,E2 -711.939} C_VEL
LIN {X 0,Y 601.418,Z 450.472,A -85,B 0,C 180,E1 -712.783,E2 -712.783} C_VEL
LIN {X 0,Y 601.377,Z 459.305,A -85,B 0,C 180,E1 -713.781,E2 -713.781} C_VEL
LIN {X 0,Y 601.362,Z 466.619,A -85,B 0,C 180,E1 -714.803,E2 -714.803} C_VEL
LIN {X 0,Y 601.346,Z 473.184,A -85,B 0,C 180,E1 -715.979,E2 -715.979} C_VEL
LIN {X 0,Y 601.378,Z 477.529,A -85,B 0,C 180,E1 -716.985,E2 -716.985} C_VEL
LIN {X 0,Y 601.343,Z 480.816,A -85,B 0,C 180,E1 -717.991,E2 -717.991} C_VEL
LIN {X 0,Y 601.348,Z 482.457,A -85,B 0,C 180,E1 -718.661,E2 -718.661} C_VEL
LIN {X 0,Y 601.339,Z 483.683,A -85,B 0,C 180,E1 -719.33,E2 -719.33} C_VEL
LIN {X 0,Y 601.336,Z 484.509,A -85,B 0,C 180,E1 -720,E2 -720} C_VEL
LIN {X 0,Y 601.348,Z 484.938,A -85,B 0,C 180,E1 -721.339,E2 -721.339} C_VEL
LIN {X 0,Y 601.341,Z 484.578,A -85,B 0,C 180,E1 -722.009,E2 -722.009} C_VEL
LIN {X 0,Y 601.321,Z 483.814,A -85,B 0,C 180,E1 -722.679,E2 -722.679} C_VEL
LIN {X 0,Y 601.341,Z 482.626,A -85,B 0,C 180,E1 -723.35,E2 -723.35} C_VEL
LIN {X 0,Y 601.332,Z 479.02,A -85,B 0,C 180,E1 -724.693,E2 -724.693} C_VEL
LIN {X 0,Y 601.373,Z 475.107,A -85,B 0,C 180,E1 -725.701,E2 -725.701} C_VEL
LIN {X 0,Y 601.36,Z 470.053,A -85,B 0,C 180,E1 -726.711,E2 -726.711} C_VEL
LIN {X 0,Y 601.388,Z 463.695,A -85,B 0,C 180,E1 -727.723,E2 -727.723} C_VEL
LIN {X 0,Y 601.407,Z 455.748,A -85,B 0,C 180,E1 -728.738,E2 -728.738} C_VEL
LIN {X 0,Y 601.421,Z 445.833,A -85,B 0,C 180,E1 -729.755,E2 -729.755} C_VEL
LIN {X 0,Y 601.466,Z 435.426,A -85,B 0,C 180,E1 -730.605,E2 -730.605} C_VEL
LIN {X 0,Y 601.499,Z 425.007,A -85,B 0,C 180,E1 -731.294,E2 -731.294} C_VEL
LIN {X 0,Y 601.538,Z 413.855,A -85,B 0,C 180,E1 -731.883,E2 -731.883} C_VEL
LIN {X 0,Y 601.573,Z 402.316,A -85,B 0,C 180,E1 -732.353,E2 -732.353} C_VEL
LIN {X 0,Y 601.44,Z 396.567,A -85,B 0,C 180,E1 -732.549,E2 -732.549} C_VEL
LIN {X 0,Y 601.42,Z 396.57,A -85,B 0,C 180,E1 -735.591,E2 -735.591} C_VEL
LIN {X 0,Y 601.396,Z 396.575,A -85,B 0,C 180,E1 -737.688,E2 -737.688} C_VEL
LIN {X 0,Y 601.432,Z 396.57,A -85,B 0,C 180,E1 -740.522,E2 -740.522} C_VEL
LIN {X 0,Y 601.397,Z 396.573,A -85,B 0,C 180,E1 -743.411,E2 -743.411} C_VEL
LIN {X 0,Y 601.422,Z 396.573,A -85,B 0,C 180,E1 -745.868,E2 -745.868} C_VEL
LIN {X 0,Y 601.44,Z 396.571,A -85,B 0,C 180,E1 -748.626,E2 -748.626} C_VEL
LIN {X 0,Y 601.423,Z 396.573,A -85,B 0,C 180,E1 -751.454,E2 -751.454} C_VEL
LIN {X 0,Y 601.43,Z 396.573,A -85,B 0,C 180,E1 -754.118,E2 -754.118} C_VEL
LIN {X 0,Y 601.441,Z 396.567,A -85,B 0,C 180,E1 -757.382,E2 -757.382} C_VEL
LIN {X 0,Y 601.407,Z 396.573,A -85,B 0,C 180,E1 -759.996,E2 -759.996} C_VEL
LIN {X 0,Y 601.418,Z 396.573,A -85,B 0,C 180,E1 -762.67,E2 -762.67} C_VEL
LIN {X 0,Y 601.401,Z 396.574,A -85,B 0,C 180,E1 -765.467,E2 -765.467} C_VEL
LIN {X 0,Y 601.424,Z 396.57,A -85,B 0,C 180,E1 -768.407,E2 -768.407} C_VEL
LIN {X 0,Y 601.443,Z 396.572,A -85,B 0,C 180,E1 -770.876,E2 -770.876} C_VEL
LIN {X 0,Y 601.446,Z 396.571,A -85,B 0,C 180,E1 -773.734,E2 -773.734} C_VEL
LIN {X 0,Y 601.447,Z 396.63,A -85,B 0,C 180,E1 -774.159,E2 -774.159} C_VEL
LIN {X 0,Y 601.684,Z 403.402,A -85,B 0,C 180,E1 -775.493,E2 -775.493} C_VEL
LIN {X 0,Y 601.755,Z 419.3,A -85,B 0,C 180,E1 -778.494,E2 -778.494} C_VEL
LIN {X 0,Y 601.692,Z 432.936,A -85,B 0,C 180,E1 -781.167,E2 -781.167} C_VEL
LIN {X 0,Y 601.638,Z 448.118,A -85,B 0,C 180,E1 -784.089,E2 -784.089} C_VEL
LIN {X 0,Y 601.585,Z 463.406,A -85,B 0,C 180,E1 -786.96,E2 -786.96} C_VEL
LIN {X 0,Y 601.525,Z 479.057,A -85,B 0,C 180,E1 -789.838,E2 -789.838} C_VEL
LIN {X 0,Y 601.487,Z 492.752,A -85,B 0,C 180,E1 -792.314,E2 -792.314} C_VEL
LIN {X 0,Y 601.437,Z 508.403,A -85,B 0,C 180,E1 -795.103,E2 -795.103} C_VEL
LIN {X 0,Y 601.413,Z 525.155,A -85,B 0,C 180,E1 -798.05,E2 -798.05} C_VEL
LIN {X 0,Y 601.591,Z 537.431,A -85,B 0,C 180,E1 -798.267,E2 -798.267} C_VEL
LIN {X 0,Y 601.561,Z 550.232,A -85,B 0,C 180,E1 -798.622,E2 -798.622} C_VEL
LIN {X 0,Y 601.539,Z 561.954,A -85,B 0,C 180,E1 -799.076,E2 -799.076} C_VEL
LIN {X 0,Y 601.482,Z 573.324,A -85,B 0,C 180,E1 -799.651,E2 -799.651} C_VEL
LIN {X 0,Y 601.467,Z 583.928,A -85,B 0,C 180,E1 -800.33,E2 -800.33} C_VEL
LIN {X 0,Y 601.435,Z 593.597,A -85,B 0,C 180,E1 -801.093,E2 -801.093} C_VEL
LIN {X 0,Y 601.407,Z 602.412,A -85,B 0,C 180,E1 -801.939,E2 -801.939} C_VEL
LIN {X 0,Y 601.388,Z 609.689,A -85,B 0,C 180,E1 -802.783,E2 -802.783} C_VEL
LIN {X 0,Y 601.375,Z 616.773,A -85,B 0,C 180,E1 -803.782,E2 -803.782} C_VEL
LIN {X 0,Y 601.373,Z 621.679,A -85,B 0,C 180,E1 -804.635,E2 -804.635} C_VEL
LIN {X 0,Y 601.353,Z 626.37,A -85,B 0,C 180,E1 -805.643,E2 -805.643} C_VEL
LIN {X 0,Y 601.345,Z 629.955,A -85,B 0,C 180,E1 -806.65,E2 -806.65} C_VEL
LIN {X 0,Y 601.325,Z 631.809,A -85,B 0,C 180,E1 -807.32,E2 -807.32} C_VEL
LIN {X 0,Y 601.341,Z 633.201,A -85,B 0,C 180,E1 -807.991,E2 -807.991} C_VEL
LIN {X 0,Y 601.339,Z 634.784,A -85,B 0,C 180,E1 -809.33,E2 -809.33} C_VEL
LIN {X 0,Y 601.335,Z 635,A -85,B 0,C 180,E1 -810,E2 -810} C_VEL
LIN {X 0,Y 601.348,Z 634.184,A -85,B 0,C 180,E1 -811.339,E2 -811.339} C_VEL
LIN {X 0,Y 601.341,Z 633.202,A -85,B 0,C 180,E1 -812.009,E2 -812.009} C_VEL
LIN {X 0,Y 601.325,Z 631.81,A -85,B 0,C 180,E1 -812.679,E2 -812.679} C_VEL
LIN {X 0,Y 601.367,Z 628.897,A -85,B 0,C 180,E1 -813.685,E2 -813.685} C_VEL
LIN {X 0,Y 601.337,Z 624.95,A -85,B 0,C 180,E1 -814.693,E2 -814.693} C_VEL
LIN {X 0,Y 601.372,Z 618.878,A -85,B 0,C 180,E1 -815.869,E2 -815.869} C_VEL
LIN {X 0,Y 601.382,Z 612.236,A -85,B 0,C 180,E1 -816.88,E2 -816.88} C_VEL
LIN {X 0,Y 601.4,Z 603.99,A -85,B 0,C 180,E1 -817.892,E2 -817.892} C_VEL
LIN {X 0,Y 601.436,Z 595.538,A -85,B 0,C 180,E1 -818.737,E2 -818.737} C_VEL
LIN {X 0,Y 601.449,Z 585.093,A -85,B 0,C 180,E1 -819.585,E2 -819.585} C_VEL
LIN {X 0,Y 601.472,Z 574.759,A -85,B 0,C 180,E1 -820.264,E2 -820.264} C_VEL
LIN {X 0,Y 601.533,Z 562.646,A -85,B 0,C 180,E1 -820.894,E2 -820.894} C_VEL
LIN {X 0,Y 601.56,Z 550.229,A -85,B 0,C 180,E1 -821.378,E2 -821.378} C_VEL
LIN {X 0,Y 601.591,Z 537.442,A -85,B 0,C 180,E1 -821.733,E2 -821.733} C_VEL
LIN {X 0,Y 601.413,Z 525.157,A -85,B 0,C 180,E1 -821.95,E2 -821.95} C_VEL
LIN {X 0,Y 601.436,Z 508.405,A -85,B 0,C 180,E1 -824.897,E2 -824.897} C_VEL
LIN {X 0,Y 601.487,Z 492.754,A -85,B 0,C 180,E1 -827.686,E2 -827.686} C_VEL
LIN {X 0,Y 601.526,Z 479.059,A -85,B 0,C 180,E1 -830.161,E2 -830.161} C_VEL
LIN {X 0,Y 601.585,Z 463.407,A -85,B 0,C 180,E1 -833.039,E2 -833.039} C_VEL
LIN {X 0,Y 601.651,Z 447.216,A -85,B 0,C 180,E1 -836.082,E2 -836.082} C_VEL
LIN {X 0,Y 601.716,Z 431.79,A -85,B 0,C 180,E1 -839.055,E2 -839.055} C_VEL
LIN {X 0,Y 601.732,Z 418.206,A -85,B 0,C 180,E1 -841.707,E2 -841.707} C_VEL
LIN {X 0,Y 601.673,Z 402.333,A -85,B 0,C 180,E1 -844.711,E2 -844.711} C_VEL
LIN {X 0,Y 601.525,Z 397.089,A -85,B 0,C 180,E1 -845.745,E2 -845.745} C_VEL
LIN {X 0,Y 601.449,Z 396.571,A -85,B 0,C 180,E1 -845.931,E2 -845.931} C_VEL
LIN {X 0,Y 601.44,Z 396.57,A -85,B 0,C 180,E1 -848.472,E2 -848.472} C_VEL
LIN {X 0,Y 601.42,Z 396.571,A -85,B 0,C 180,E1 -850.874,E2 -850.874} C_VEL
LIN {X 0,Y 601.43,Z 396.573,A -85,B 0,C 180,E1 -853.586,E2 -853.586} C_VEL
LIN {X 0,Y 601.452,Z 396.567,A -85,B 0,C 180,E1 -856.425,E2 -856.425} C_VEL
LIN {X 0,Y 601.418,Z 396.572,A -85,B 0,C 180,E1 -859.426,E2 -859.426} C_VEL
LIN {X 0,Y 601.425,Z 396.57,A -85,B 0,C 180,E1 -861.732,E2 -861.732} C_VEL
LIN {X 0,Y 601.398,Z 396.575,A -85,B 0,C 180,E1 -864.246,E2 -864.246} C_VEL
LIN {X 0,Y 601.421,Z 396.573,A -85,B 0,C 180,E1 -866.686,E2 -866.686} C_VEL
LIN {X 0,Y 601.417,Z 396.572,A -85,B 0,C 180,E1 -869.058,E2 -869.058} C_VEL
LIN {X 0,Y 601.435,Z 396.569,A -85,B 0,C 180,E1 -871.373,E2 -871.373} C_VEL
LIN {X 0,Y 601.411,Z 396.572,A -85,B 0,C 180,E1 -873.637,E2 -873.637} C_VEL
LIN {X 0,Y 601.422,Z 396.572,A -85,B 0,C 180,E1 -876.59,E2 -876.59} C_VEL
LIN {X 0,Y 601.43,Z 396.571,A -85,B 0,C 180,E1 -879.478,E2 -879.478} C_VEL
LIN {X 0,Y 601.401,Z 396.574,A -85,B 0,C 180,E1 -882.312,E2 -882.312} C_VEL
LIN {X 0,Y 601.423,Z 396.571,A -85,B 0,C 180,E1 -884.409,E2 -884.409} C_VEL
LIN {X 0,Y 601.427,Z 396.573,A -85,B 0,C 180,E1 -887.172,E2 -887.172} C_VEL
LIN {X 0,Y 601.432,Z 396.57,A -85,B 0,C 180,E1 -889.905,E2 -889.905} C_VEL
LIN {X 0,Y 601.44,Z 396.572,A -85,B 0,C 180,E1 -892.615,E2 -892.615} C_VEL
LIN {X 0,Y 601.429,Z 396.57,A -85,B 0,C 180,E1 -895.308,E2 -895.308} C_VEL
LIN {X 0,Y 601.438,Z 396.572,A -85,B 0,C 180,E1 -897.991,E2 -897.991} C_VEL
LIN {X 0,Y 601.455,Z 396.567,A -85,B 0,C 180,E1 -900.67,E2 -900.67} C_VEL
LIN {X 0,Y 601.429,Z 396.572,A -85,B 0,C 180,E1 -903.35,E2 -903.35} C_VEL
LIN {X 0,Y 601.412,Z 396.572,A -85,B 0,C 180,E1 -906.037,E2 -906.037} C_VEL
LIN {X 0,Y 601.442,Z 396.57,A -85,B 0,C 180,E1 -908.738,E2 -908.738} C_VEL
LIN {X 0,Y 601.437,Z 396.569,A -85,B 0,C 180,E1 -911.458,E2 -911.458} C_VEL
LIN {X 0,Y 601.412,Z 396.573,A -85,B 0,C 180,E1 -912.38,E2 -912.38} C_VEL
LIN {X 0,Y 600.75,Z 396.656,A -85,B 0,C 180,E1 -912.939,E2 -912.939} C_VEL
LIN {X 0,Y 597.9,Z 397.01,A -85,B 0,C 180,E1 -913.847,E2 -913.847} C_VEL
LIN {X 0,Y 595.487,Z 397.311,A -85,B 0,C 180,E1 -914.577,E2 -914.577} C_VEL
LIN {X 0,Y 594.448,Z 397.44,A -85,B 0,C 180,E1 -915.141,E2 -915.141} C_VEL
LIN {X 0,Y 594.361,Z 397.449,A -85,B 0,C 180,E1 -915.332,E2 -915.332} C_VEL
LIN {X 0,Y 594.392,Z 397.447,A -85,B 0,C 180,E1 -917.193,E2 -917.193} C_VEL
LIN {X 0,Y 594.38,Z 397.448,A -85,B 0,C 180,E1 -920.054,E2 -920.054} C_VEL
LIN {X 0,Y 594.368,Z 397.452,A -85,B 0,C 180,E1 -922.967,E2 -922.967} C_VEL
LIN {X 0,Y 594.379,Z 397.451,A -85,B 0,C 180,E1 -925.193,E2 -925.193} C_VEL
LIN {X 0,Y 594.389,Z 397.448,A -85,B 0,C 180,E1 -927.527,E2 -927.527} C_VEL
LIN {X 0,Y 594.388,Z 397.448,A -85,B 0,C 180,E1 -930.328,E2 -930.328} C_VEL
LIN {X 0,Y 594.383,Z 397.449,A -85,B 0,C 180,E1 -932.95,E2 -932.95} C_VEL
LIN {X 0,Y 594.36,Z 397.45,A -85,B 0,C 180,E1 -935.409,E2 -935.409} C_VEL
LIN {X 0,Y 594.391,Z 397.448,A -85,B 0,C 180,E1 -937.941,E2 -937.941} C_VEL
LIN {X 0,Y 594.378,Z 397.448,A -85,B 0,C 180,E1 -940.822,E2 -940.822} C_VEL
LIN {X 0,Y 594.386,Z 397.448,A -85,B 0,C 180,E1 -943.841,E2 -943.841} C_VEL
LIN {X 0,Y 594.384,Z 397.45,A -85,B 0,C 180,E1 -946.702,E2 -946.702} C_VEL
LIN {X 0,Y 594.372,Z 397.449,A -85,B 0,C 180,E1 -949.433,E2 -949.433} C_VEL
LIN {X 0,Y 594.391,Z 397.448,A -85,B 0,C 180,E1 -952.392,E2 -952.392} C_VEL
LIN {X 0,Y 594.403,Z 397.448,A -85,B 0,C 180,E1 -955.422,E2 -955.422} C_VEL
LIN {X 0,Y 594.398,Z 397.446,A -85,B 0,C 180,E1 -958.355,E2 -958.355} C_VEL
LIN {X 0,Y 594.387,Z 397.449,A -85,B 0,C 180,E1 -961.042,E2 -961.042} C_VEL
LIN {X 0,Y 594.387,Z 397.449,A -85,B 0,C 180,E1 -963.978,E2 -963.978} C_VEL
LIN {X 0,Y 594.392,Z 397.449,A -85,B 0,C 180,E1 -966.296,E2 -966.296} C_VEL
LIN {X 0,Y 594.411,Z 397.445,A -85,B 0,C 180,E1 -969.225,E2 -969.225} C_VEL
LIN {X 0,Y 594.386,Z 397.448,A -85,B 0,C 180,E1 -972.096,E2 -972.096} C_VEL
LIN {X 0,Y 594.375,Z 397.452,A -85,B 0,C 180,E1 -974.922,E2 -974.922} C_VEL
LIN {X 0,Y 594.392,Z 397.446,A -85,B 0,C 180,E1 -977.712,E2 -977.712} C_VEL
LIN {X 0,Y 594.374,Z 397.451,A -85,B 0,C 180,E1 -980.472,E2 -980.472} C_VEL
LIN {X 0,Y 594.394,Z 397.451,A -85,B 0,C 180,E1 -981.437,E2 -981.437} C_VEL
LIN {X 0,Y 594.573,Z 408.627,A -85,B 0,C 180,E1 -981.846,E2 -981.846} C_VEL
LIN {X 0,Y 594.527,Z 420.984,A -85,B 0,C 180,E1 -982.443,E2 -982.443} C_VEL
LIN {X 0,Y 594.447,Z 432.017,A -85,B 0,C 180,E1 -983.125,E2 -983.125} C_VEL
LIN {X 0,Y 594.402,Z 442.013,A -85,B 0,C 180,E1 -983.892,E2 -983.892} C_VEL
LIN {X 0,Y 594.379,Z 451.03,A -85,B 0,C 180,E1 -984.742,E2 -984.742} C_VEL
LIN {X 0,Y 594.346,Z 459.851,A -85,B 0,C 180,E1 -985.762,E2 -985.762} C_VEL
LIN {X 0,Y 594.321,Z 466.937,A -85,B 0,C 180,E1 -986.78,E2 -986.78} C_VEL
LIN {X 0,Y 594.258,Z 473.421,A -85,B 0,C 180,E1 -987.967,E2 -987.967} C_VEL
LIN {X 0,Y 594.25,Z 477.71,A -85,B 0,C 180,E1 -988.984,E2 -988.984} C_VEL
LIN {X 0,Y 594.238,Z 480.946,A -85,B 0,C 180,E1 -990,E2 -990} C_VEL
LIN {X 0,Y 594.249,Z 483.758,A -85,B 0,C 180,E1 -991.356,E2 -991.356} C_VEL
LIN {X 0,Y 594.241,Z 484.555,A -85,B 0,C 180,E1 -992.033,E2 -992.033} C_VEL
LIN {X 0,Y 594.258,Z 484.927,A -85,B 0,C 180,E1 -993.39,E2 -993.39} C_VEL
LIN {X 0,Y 594.254,Z 484.546,A -85,B 0,C 180,E1 -994.069,E2 -994.069} C_VEL
LIN {X 0,Y 594.227,Z 483.736,A -85,B 0,C 180,E1 -994.749,E2 -994.749} C_VEL
LIN {X 0,Y 594.263,Z 482.51,A -85,B 0,C 180,E1 -995.429,E2 -995.429} C_VEL
LIN {X 0,Y 594.263,Z 479.527,A -85,B 0,C 180,E1 -996.574,E2 -996.574} C_VEL
LIN {X 0,Y 594.281,Z 474.849,A -85,B 0,C 180,E1 -997.817,E2 -997.817} C_VEL
LIN {X 0,Y 594.292,Z 468.699,A -85,B 0,C 180,E1 -999.015,E2 -999.015} C_VEL
LIN {X 0,Y 594.327,Z 461.961,A -85,B 0,C 180,E1 -1000.045,E2 -1000.045} C_VEL
LIN {X 0,Y 594.336,Z 453.864,A -85,B 0,C 180,E1 -1001.045,E2 -1001.045} C_VEL
LIN {X 0,Y 594.395,Z 444.916,A -85,B 0,C 180,E1 -1001.942,E2 -1001.942} C_VEL
LIN {X 0,Y 594.425,Z 434.232,A -85,B 0,C 180,E1 -1002.808,E2 -1002.808} C_VEL
LIN {X 0,Y 594.473,Z 423.582,A -85,B 0,C 180,E1 -1003.503,E2 -1003.503} C_VEL
LIN {X 0,Y 594.542,Z 412.024,A -85,B 0,C 180,E1 -1004.096,E2 -1004.096} C_VEL
LIN {X 0,Y 594.616,Z 399.216,A -85,B 0,C 180,E1 -1004.59,E2 -1004.59} C_VEL
LIN {X 0,Y 594.395,Z 397.447,A -85,B 0,C 180,E1 -1004.661,E2 -1004.661} C_VEL
LIN {X 0,Y 594.383,Z 397.441,A -85,B 0,C 180,E1 -1007.194,E2 -1007.194} C_VEL
LIN {X 0,Y 594.376,Z 397.446,A -85,B 0,C 180,E1 -1010.054,E2 -1010.054} C_VEL
LIN {X 0,Y 594.362,Z 397.444,A -85,B 0,C 180,E1 -1012.968,E2 -1012.968} C_VEL
LIN {X 0,Y 594.378,Z 397.441,A -85,B 0,C 180,E1 -1015.193,E2 -1015.193} C_VEL
LIN {X 0,Y 594.373,Z 397.442,A -85,B 0,C 180,E1 -1017.523,E2 -1017.523} C_VEL
LIN {X 0,Y 594.392,Z 397.448,A -85,B 0,C 180,E1 -1020.328,E2 -1020.328} C_VEL
LIN {X 0,Y 594.38,Z 397.441,A -85,B 0,C 180,E1 -1022.95,E2 -1022.95} C_VEL
LIN {X 0,Y 594.364,Z 397.443,A -85,B 0,C 180,E1 -1025.408,E2 -1025.408} C_VEL
LIN {X 0,Y 594.394,Z 397.445,A -85,B 0,C 180,E1 -1027.94,E2 -1027.94} C_VEL
LIN {X 0,Y 594.379,Z 397.441,A -85,B 0,C 180,E1 -1030.822,E2 -1030.822} C_VEL
LIN {X 0,Y 594.373,Z 397.447,A -85,B 0,C 180,E1 -1033.84,E2 -1033.84} C_VEL
LIN {X 0,Y 594.385,Z 397.441,A -85,B 0,C 180,E1 -1036.702,E2 -1036.702} C_VEL
LIN {X 0,Y 594.373,Z 397.443,A -85,B 0,C 180,E1 -1039.433,E2 -1039.433} C_VEL
LIN {X 0,Y 594.394,Z 397.442,A -85,B 0,C 180,E1 -1042.392,E2 -1042.392} C_VEL
LIN {X 0,Y 594.38,Z 397.443,A -85,B 0,C 180,E1 -1045.42,E2 -1045.42} C_VEL
LIN {X 0,Y 594.382,Z 397.443,A -85,B 0,C 180,E1 -1048.357,E2 -1048.357} C_VEL
LIN {X 0,Y 594.387,Z 397.44,A -85,B 0,C 180,E1 -1051.042,E2 -1051.042} C_VEL
LIN {X 0,Y 594.388,Z 397.447,A -85,B 0,C 180,E1 -1053.978,E2 -1053.978} C_VEL
LIN {X 0,Y 594.377,Z 397.444,A -85,B 0,C 180,E1 -1056.295,E2 -1056.295} C_VEL
LIN {X 0,Y 594.406,Z 397.439,A -85,B 0,C 180,E1 -1059.224,E2 -1059.224} C_VEL
LIN {X 0,Y 594.355,Z 397.448,A -85,B 0,C 180,E1 -1062.095,E2 -1062.095} C_VEL
LIN {X 0,Y 594.367,Z 397.445,A -85,B 0,C 180,E1 -1064.219,E2 -1064.219} C_VEL
LIN {X 0,Y 594.381,Z 397.442,A -85,B 0,C 180,E1 -1066.321,E2 -1066.321} C_VEL
LIN {X 0,Y 594.378,Z 397.444,A -85,B 0,C 180,E1 -1069.095,E2 -1069.095} C_VEL
LIN {X 0,Y 594.411,Z 397.538,A -85,B 0,C 180,E1 -1069.44,E2 -1069.44} C_VEL
LIN {X 0,Y 594.569,Z 409.22,A -85,B 0,C 180,E1 -1069.873,E2 -1069.873} C_VEL
LIN {X 0,Y 594.495,Z 421.53,A -85,B 0,C 180,E1 -1070.473,E2 -1070.473} C_VEL
LIN {X 0,Y 594.446,Z 432.527,A -85,B 0,C 180,E1 -1071.159,E2 -1071.159} C_VEL
LIN {X 0,Y 594.431,Z 441.439,A -85,B 0,C 180,E1 -1071.843,E2 -1071.843} C_VEL
LIN {X 0,Y 594.359,Z 450.585,A -85,B 0,C 180,E1 -1072.697,E2 -1072.697} C_VEL
LIN {X 0,Y 594.331,Z 458.49,A -85,B 0,C 180,E1 -1073.592,E2 -1073.592} C_VEL
LIN {X 0,Y 594.296,Z 465.582,A -85,B 0,C 180,E1 -1074.571,E2 -1074.571} C_VEL
LIN {X 0,Y 594.278,Z 471.548,A -85,B 0,C 180,E1 -1075.591,E2 -1075.591} C_VEL
LIN {X 0,Y 594.271,Z 476.265,A -85,B 0,C 180,E1 -1076.61,E2 -1076.61} C_VEL
LIN {X 0,Y 594.256,Z 479.876,A -85,B 0,C 180,E1 -1077.628,E2 -1077.628} C_VEL
LIN {X 0,Y 594.248,Z 482.485,A -85,B 0,C 180,E1 -1078.645,E2 -1078.645} C_VEL
LIN {X 0,Y 594.239,Z 483.701,A -85,B 0,C 180,E1 -1079.322,E2 -1079.322} C_VEL
LIN {X 0,Y 594.237,Z 484.513,A -85,B 0,C 180,E1 -1080,E2 -1080} C_VEL
LIN {X 0,Y 594.239,Z 484.923,A -85,B 0,C 180,E1 -1080.678,E2 -1080.678} C_VEL
LIN {X 0,Y 594.239,Z 484.562,A -85,B 0,C 180,E1 -1082.033,E2 -1082.033} C_VEL
LIN {X 0,Y 594.222,Z 483.792,A -85,B 0,C 180,E1 -1082.712,E2 -1082.712} C_VEL
LIN {X 0,Y 594.26,Z 482.602,A -85,B 0,C 180,E1 -1083.39,E2 -1083.39} C_VEL
LIN {X 0,Y 594.234,Z 478.979,A -85,B 0,C 180,E1 -1084.749,E2 -1084.749} C_VEL
LIN {X 0,Y 594.299,Z 475.053,A -85,B 0,C 180,E1 -1085.769,E2 -1085.769} C_VEL
LIN {X 0,Y 594.28,Z 469.975,A -85,B 0,C 180,E1 -1086.792,E2 -1086.792} C_VEL
LIN {X 0,Y 594.305,Z 463.601,A -85,B 0,C 180,E1 -1087.816,E2 -1087.816} C_VEL
LIN {X 0,Y 594.352,Z 455.641,A -85,B 0,C 180,E1 -1088.843,E2 -1088.843} C_VEL
LIN {X 0,Y 594.39,Z 447.506,A -85,B 0,C 180,E1 -1089.7,E2 -1089.7} C_VEL
LIN {X 0,Y 594.436,Z 437.549,A -85,B 0,C 180,E1 -1090.559,E2 -1090.559} C_VEL
LIN {X 0,Y 594.462,Z 426.585,A -85,B 0,C 180,E1 -1091.32,E2 -1091.32} C_VEL
LIN {X 0,Y 594.568,Z 415.355,A -85,B 0,C 180,E1 -1091.938,E2 -1091.938} C_VEL
LIN {X 0,Y 594.595,Z 403.178,A -85,B 0,C 180,E1 -1092.457,E2 -1092.457} C_VEL
LIN {X 0,Y 594.402,Z 397.444,A -85,B 0,C 180,E1 -1092.657,E2 -1092.657} C_VEL
LIN {X 0,Y 594.38,Z 397.447,A -85,B 0,C 180,E1 -1095.078,E2 -1095.078} C_VEL
LIN {X 0,Y 594.387,Z 397.448,A -85,B 0,C 180,E1 -1097.193,E2 -1097.193} C_VEL
LIN {X 0,Y 594.378,Z 397.45,A -85,B 0,C 180,E1 -1100.054,E2 -1100.054} C_VEL
LIN {X 0,Y 594.361,Z 397.453,A -85,B 0,C 180,E1 -1102.967,E2 -1102.967} C_VEL
LIN {X 0,Y 594.38,Z 397.446,A -85,B 0,C 180,E1 -1105.193,E2 -1105.193} C_VEL
LIN {X 0,Y 594.39,Z 397.446,A -85,B 0,C 180,E1 -1107.527,E2 -1107.527} C_VEL
LIN {X 0,Y 594.39,Z 397.446,A -85,B 0,C 180,E1 -1110.328,E2 -1110.328} C_VEL
LIN {X 0,Y 594.383,Z 397.448,A -85,B 0,C 180,E1 -1112.95,E2 -1112.95} C_VEL
LIN {X 0,Y 594.353,Z 397.453,A -85,B 0,C 180,E1 -1115.409,E2 -1115.409} C_VEL
LIN {X 0,Y 594.386,Z 397.446,A -85,B 0,C 180,E1 -1117.941,E2 -1117.941} C_VEL
LIN {X 0,Y 594.379,Z 397.448,A -85,B 0,C 180,E1 -1120.822,E2 -1120.822} C_VEL
LIN {X 0,Y 594.388,Z 397.45,A -85,B 0,C 180,E1 -1123.841,E2 -1123.841} C_VEL
LIN {X 0,Y 594.37,Z 397.452,A -85,B 0,C 180,E1 -1126.7,E2 -1126.7} C_VEL
LIN {X 0,Y 594.372,Z 397.452,A -85,B 0,C 180,E1 -1129.433,E2 -1129.433} C_VEL
LIN {X 0,Y 594.392,Z 397.449,A -85,B 0,C 180,E1 -1132.392,E2 -1132.392} C_VEL
LIN {X 0,Y 594.428,Z 397.523,A -85,B 0,C 180,E1 -1133.97,E2 -1133.97} C_VEL
LIN {X 0,Y 594.779,Z 402.8,A -85,B 0,C 180,E1 -1135.034,E2 -1135.034} C_VEL
LIN {X 0,Y 594.788,Z 418.901,A -85,B 0,C 180,E1 -1138.127,E2 -1138.127} C_VEL
LIN {X 0,Y 594.85,Z 430.146,A -85,B 0,C 180,E1 -1140.25,E2 -1140.25} C_VEL
LIN {X 0,Y 594.735,Z 443.841,A -85,B 0,C 180,E1 -1142.938,E2 -1142.938} C_VEL
LIN {X 0,Y 594.632,Z 457.536,A -85,B 0,C 180,E1 -1145.564,E2 -1145.564} C_VEL
LIN {X 0,Y 594.58,Z 471.231,A -85,B 0,C 180,E1 -1148.14,E2 -1148.14} C_VEL
LIN {X 0,Y 594.521,Z 486.904,A -85,B 0,C 180,E1 -1151.033,E2 -1151.033} C_VEL
LIN {X 0,Y 594.411,Z 502.534,A -85,B 0,C 180,E1 -1153.868,E2 -1153.868} C_VEL
LIN {X 0,Y 594.363,Z 518.186,A -85,B 0,C 180,E1 -1156.669,E2 -1156.669} C_VEL
LIN {X 0,Y 594.356,Z 525.155,A -85,B 0,C 180,E1 -1157.906,E2 -1157.906} C_VEL
LIN {X 0,Y 594.673,Z 530.936,A -85,B 0,C 180,E1 -1157.999,E2 -1157.999} C_VEL
LIN {X 0,Y 594.623,Z 544.21,A -85,B 0,C 180,E1 -1158.301,E2 -1158.301} C_VEL
LIN {X 0,Y 594.563,Z 557.245,A -85,B 0,C 180,E1 -1158.744,E2 -1158.744} C_VEL
LIN {X 0,Y 594.525,Z 568.629,A -85,B 0,C 180,E1 -1159.27,E2 -1159.27} C_VEL
LIN {X 0,Y 594.469,Z 580.197,A -85,B 0,C 180,E1 -1159.957,E2 -1159.957} C_VEL
LIN {X 0,Y 594.414,Z 590.593,A -85,B 0,C 180,E1 -1160.729,E2 -1160.729} C_VEL
LIN {X 0,Y 594.383,Z 599.11,A -85,B 0,C 180,E1 -1161.5,E2 -1161.5} C_VEL
LIN {X 0,Y 594.347,Z 606.959,A -85,B 0,C 180,E1 -1162.355,E2 -1162.355} C_VEL
LIN {X 0,Y 594.283,Z 614.812,A -85,B 0,C 180,E1 -1163.408,E2 -1163.408} C_VEL
LIN {X 0,Y 594.289,Z 621.679,A -85,B 0,C 180,E1 -1164.571,E2 -1164.571} C_VEL
LIN {X 0,Y 594.27,Z 626.37,A -85,B 0,C 180,E1 -1165.591,E2 -1165.591} C_VEL
LIN {X 0,Y 594.267,Z 629.956,A -85,B 0,C 180,E1 -1166.61,E2 -1166.61} C_VEL
LIN {X 0,Y 594.226,Z 631.808,A -85,B 0,C 180,E1 -1167.288,E2 -1167.288} C_VEL
LIN {X 0,Y 594.24,Z 633.201,A -85,B 0,C 180,E1 -1167.967,E2 -1167.967} C_VEL
LIN {X 0,Y 594.239,Z 634.784,A -85,B 0,C 180,E1 -1169.322,E2 -1169.322} C_VEL
LIN {X 0,Y 594.236,Z 635,A -85,B 0,C 180,E1 -1170,E2 -1170} C_VEL
LIN {X 0,Y 594.247,Z 634.185,A -85,B 0,C 180,E1 -1171.355,E2 -1171.355} C_VEL
LIN {X 0,Y 594.24,Z 633.202,A -85,B 0,C 180,E1 -1172.033,E2 -1172.033} C_VEL
LIN {X 0,Y 594.226,Z 631.81,A -85,B 0,C 180,E1 -1172.711,E2 -1172.711} C_VEL
LIN {X 0,Y 594.288,Z 628.896,A -85,B 0,C 180,E1 -1173.729,E2 -1173.729} C_VEL
LIN {X 0,Y 594.242,Z 624.95,A -85,B 0,C 180,E1 -1174.749,E2 -1174.749} C_VEL
LIN {X 0,Y 594.304,Z 618.878,A -85,B 0,C 180,E1 -1175.939,E2 -1175.939} C_VEL
LIN {X 0,Y 594.308,Z 612.237,A -85,B 0,C 180,E1 -1176.962,E2 -1176.962} C_VEL
LIN {X 0,Y 594.359,Z 603.991,A -85,B 0,C 180,E1 -1177.986,E2 -1177.986} C_VEL
LIN {X 0,Y 594.382,Z 595.538,A -85,B 0,C 180,E1 -1178.842,E2 -1178.842} C_VEL
LIN {X 0,Y 594.431,Z 585.095,A -85,B 0,C 180,E1 -1179.699,E2 -1179.699} C_VEL
LIN {X 0,Y 594.482,Z 574.76,A -85,B 0,C 180,E1 -1180.386,E2 -1180.386} C_VEL
LIN {X 0,Y 594.532,Z 563.76,A -85,B 0,C 180,E1 -1180.972,E2 -1180.972} C_VEL
LIN {X 0,Y 594.582,Z 551.724,A -85,B 0,C 180,E1 -1181.464,E2 -1181.464} C_VEL
LIN {X 0,Y 594.629,Z 538.356,A -85,B 0,C 180,E1 -1181.85,E2 -1181.85} C_VEL
LIN {X 0,Y 594.577,Z 526.608,A -85,B 0,C 180,E1 -1182.068,E2 -1182.068} C_VEL
LIN {X 0,Y 594.361,Z 525.035,A -85,B 0,C 180,E1 -1182.115,E2 -1182.115} C_VEL
LIN {X 0,Y 594.395,Z 510.362,A -85,B 0,C 180,E1 -1184.727,E2 -1184.727} C_VEL
LIN {X 0,Y 594.463,Z 494.71,A -85,B 0,C 180,E1 -1187.546,E2 -1187.546} C_VEL
LIN {X 0,Y 594.543,Z 481.015,A -85,B 0,C 180,E1 -1190.048,E2 -1190.048} C_VEL
LIN {X 0,Y 594.621,Z 465.364,A -85,B 0,C 180,E1 -1192.957,E2 -1192.957} C_VEL
LIN {X 0,Y 594.697,Z 449.712,A -85,B 0,C 180,E1 -1195.929,E2 -1195.929} C_VEL
LIN {X 0,Y 594.8,Z 436.017,A -85,B 0,C 180,E1 -1198.59,E2 -1198.59} C_VEL
LIN {X 0,Y 594.835,Z 425.005,A -85,B 0,C 180,E1 -1200.73,E2 -1200.73} C_VEL
LIN {X 0,Y 594.714,Z 410.114,A -85,B 0,C 180,E1 -1203.536,E2 -1203.536} C_VEL
LIN {X 0,Y 594.731,Z 399.677,A -85,B 0,C 180,E1 -1205.59,E2 -1205.59} C_VEL
LIN {X 0,Y 594.423,Z 397.446,A -85,B 0,C 180,E1 -1206.082,E2 -1206.082} C_VEL
LIN {X 0,Y 594.392,Z 397.447,A -85,B 0,C 180,E1 -1208.804,E2 -1208.804} C_VEL
LIN {X 0,Y 594.384,Z 397.448,A -85,B 0,C 180,E1 -1211.848,E2 -1211.848} C_VEL
LIN {X 0,Y 594.366,Z 397.452,A -85,B 0,C 180,E1 -1214.809,E2 -1214.809} C_VEL
LIN {X 0,Y 594.373,Z 397.449,A -85,B 0,C 180,E1 -1217.625,E2 -1217.625} C_VEL
LIN {X 0,Y 594.395,Z 397.448,A -85,B 0,C 180,E1 -1220.321,E2 -1220.321} C_VEL
LIN {X 0,Y 594.388,Z 397.447,A -85,B 0,C 180,E1 -1222.913,E2 -1222.913} C_VEL
LIN {X 0,Y 594.383,Z 397.448,A -85,B 0,C 180,E1 -1225.861,E2 -1225.861} C_VEL
LIN {X 0,Y 594.372,Z 397.451,A -85,B 0,C 180,E1 -1228.65,E2 -1228.65} C_VEL
LIN {X 0,Y 594.386,Z 397.45,A -85,B 0,C 180,E1 -1231.042,E2 -1231.042} C_VEL
LIN {X 0,Y 594.395,Z 397.447,A -85,B 0,C 180,E1 -1233.976,E2 -1233.976} C_VEL
LIN {X 0,Y 594.392,Z 397.449,A -85,B 0,C 180,E1 -1236.296,E2 -1236.296} C_VEL
LIN {X 0,Y 594.404,Z 397.445,A -85,B 0,C 180,E1 -1239.224,E2 -1239.224} C_VEL
LIN {X 0,Y 594.357,Z 397.452,A -85,B 0,C 180,E1 -1242.095,E2 -1242.095} C_VEL
LIN {X 0,Y 594.376,Z 397.449,A -85,B 0,C 180,E1 -1244.219,E2 -1244.219} C_VEL
LIN {X 0,Y 594.374,Z 397.45,A -85,B 0,C 180,E1 -1247.017,E2 -1247.017} C_VEL
LIN {X 0,Y 594.394,Z 397.447,A -85,B 0,C 180,E1 -1249.784,E2 -1249.784} C_VEL
LIN {X 0,Y 594.394,Z 397.449,A -85,B 0,C 180,E1 -1252.527,E2 -1252.527} C_VEL
LIN {X 0,Y 594.398,Z 397.446,A -85,B 0,C 180,E1 -1255.253,E2 -1255.253} C_VEL
LIN {X 0,Y 594.407,Z 397.447,A -85,B 0,C 180,E1 -1257.967,E2 -1257.967} C_VEL
LIN {X 0,Y 594.426,Z 397.442,A -85,B 0,C 180,E1 -1260.678,E2 -1260.678} C_VEL
LIN {X 0,Y 594.38,Z 397.45,A -85,B 0,C 180,E1 -1263.389,E2 -1263.389} C_VEL
LIN {X 0,Y 594.368,Z 397.45,A -85,B 0,C 180,E1 -1266.109,E2 -1266.109} C_VEL
LIN {X 0,Y 594.403,Z 397.448,A -85,B 0,C 180,E1 -1268.842,E2 -1268.842} C_VEL
LIN {X 0,Y 594.396,Z 397.446,A -85,B 0,C 180,E1 -1271.596,E2 -1271.596} C_VEL
LIN {X 0,Y 594.393,Z 397.449,A -85,B 0,C 180,E1 -1274.377,E2 -1274.377} C_VEL
LIN {X 0,Y 594.361,Z 397.449,A -85,B 0,C 180,E1 -1275.332,E2 -1275.332} C_VEL
LIN {X 0,Y 593.687,Z 397.535,A -85,B 0,C 180,E1 -1275.898,E2 -1275.898} C_VEL
LIN {X 0,Y 590.821,Z 397.891,A -85,B 0,C 180,E1 -1276.816,E2 -1276.816} C_VEL
LIN {X 0,Y 588.412,Z 398.194,A -85,B 0,C 180,E1 -1277.554,E2 -1277.554} C_VEL
LIN {X 0,Y 587.391,Z 398.319,A -85,B 0,C 180,E1 -1278.125,E2 -1278.125} C_VEL
LIN {X 0,Y 587.314,Z 398.327,A -85,B 0,C 180,E1 -1278.318,E2 -1278.318} C_VEL
LIN {X 0,Y 587.362,Z 398.323,A -85,B 0,C 180,E1 -1281.045,E2 -1281.045} C_VEL
LIN {X 0,Y 587.342,Z 398.328,A -85,B 0,C 180,E1 -1284.006,E2 -1284.006} C_VEL
LIN {X 0,Y 587.341,Z 398.327,A -85,B 0,C 180,E1 -1286.279,E2 -1286.279} C_VEL
LIN {X 0,Y 587.353,Z 398.323,A -85,B 0,C 180,E1 -1289.134,E2 -1289.134} C_VEL
LIN {X 0,Y 587.35,Z 398.325,A -85,B 0,C 180,E1 -1291.836,E2 -1291.836} C_VEL
LIN {X 0,Y 587.354,Z 398.323,A -85,B 0,C 180,E1 -1294.348,E2 -1294.348} C_VEL
LIN {X 0,Y 587.357,Z 398.323,A -85,B 0,C 180,E1 -1296.747,E2 -1296.747} C_VEL
LIN {X 0,Y 587.334,Z 398.327,A -85,B 0,C 180,E1 -1299.361,E2 -1299.361} C_VEL
LIN {X 0,Y 587.338,Z 398.326,A -85,B 0,C 180,E1 -1302.108,E2 -1302.108} C_VEL
LIN {X 0,Y 587.32,Z 398.327,A -85,B 0,C 180,E1 -1305.089,E2 -1305.089} C_VEL
LIN {X 0,Y 587.357,Z 398.325,A -85,B 0,C 180,E1 -1307.928,E2 -1307.928} C_VEL
LIN {X 0,Y 587.337,Z 398.327,A -85,B 0,C 180,E1 -1311.058,E2 -1311.058} C_VEL
LIN {X 0,Y 587.352,Z 398.326,A -85,B 0,C 180,E1 -1313.293,E2 -1313.293} C_VEL
LIN {X 0,Y 587.373,Z 398.321,A -85,B 0,C 180,E1 -1315.781,E2 -1315.781} C_VEL
LIN {X 0,Y 587.359,Z 398.323,A -85,B 0,C 180,E1 -1318.232,E2 -1318.232} C_VEL
LIN {X 0,Y 587.355,Z 398.326,A -85,B 0,C 180,E1 -1320.867,E2 -1320.867} C_VEL
LIN {X 0,Y 587.362,Z 398.323,A -85,B 0,C 180,E1 -1323.82,E2 -1323.82} C_VEL
LIN {X 0,Y 587.34,Z 398.326,A -85,B 0,C 180,E1 -1325.994,E2 -1325.994} C_VEL
LIN {X 0,Y 587.327,Z 398.328,A -85,B 0,C 180,E1 -1328.226,E2 -1328.226} C_VEL
LIN {X 0,Y 587.352,Z 398.323,A -85,B 0,C 180,E1 -1331.151,E2 -1331.151} C_VEL
LIN {X 0,Y 587.334,Z 398.326,A -85,B 0,C 180,E1 -1333.311,E2 -1333.311} C_VEL
LIN {X 0,Y 587.363,Z 398.324,A -85,B 0,C 180,E1 -1336.154,E2 -1336.154} C_VEL
LIN {X 0,Y 587.347,Z 398.325,A -85,B 0,C 180,E1 -1338.963,E2 -1338.963} C_VEL
LIN {X 0,Y 587.333,Z 398.328,A -85,B 0,C 180,E1 -1341.311,E2 -1341.311} C_VEL
LIN {X 0,Y 587.666,Z 401.691,A -85,B 0,C 180,E1 -1341.446,E2 -1341.446} C_VEL
LIN {X 0,Y 587.593,Z 413.323,A -85,B 0,C 180,E1 -1341.921,E2 -1341.921} C_VEL
LIN {X 0,Y 587.524,Z 424.625,A -85,B 0,C 180,E1 -1342.525,E2 -1342.525} C_VEL
LIN {X 0,Y 587.409,Z 436.361,A -85,B 0,C 180,E1 -1343.324,E2 -1343.324} C_VEL
LIN {X 0,Y 587.34,Z 446.241,A -85,B 0,C 180,E1 -1344.163,E2 -1344.163} C_VEL
LIN {X 0,Y 587.287,Z 455.997,A -85,B 0,C 180,E1 -1345.195,E2 -1345.195} C_VEL
LIN {X 0,Y 587.232,Z 463.844,A -85,B 0,C 180,E1 -1346.226,E2 -1346.226} C_VEL
LIN {X 0,Y 587.168,Z 470.117,A -85,B 0,C 180,E1 -1347.256,E2 -1347.256} C_VEL
LIN {X 0,Y 587.204,Z 475.121,A -85,B 0,C 180,E1 -1348.286,E2 -1348.286} C_VEL
LIN {X 0,Y 587.145,Z 479.039,A -85,B 0,C 180,E1 -1349.314,E2 -1349.314} C_VEL
LIN {X 0,Y 587.14,Z 481.043,A -85,B 0,C 180,E1 -1350,E2 -1350} C_VEL
LIN {X 0,Y 587.139,Z 482.622,A -85,B 0,C 180,E1 -1350.686,E2 -1350.686} C_VEL
LIN {X 0,Y 587.149,Z 483.801,A -85,B 0,C 180,E1 -1351.372,E2 -1351.372} C_VEL
LIN {X 0,Y 587.14,Z 484.581,A -85,B 0,C 180,E1 -1352.058,E2 -1352.058} C_VEL
LIN {X 0,Y 587.181,Z 484.919,A -85,B 0,C 180,E1 -1353.431,E2 -1353.431} C_VEL
LIN {X 0,Y 587.17,Z 484.515,A -85,B 0,C 180,E1 -1354.118,E2 -1354.118} C_VEL
LIN {X 0,Y 587.127,Z 483.678,A -85,B 0,C 180,E1 -1354.807,E2 -1354.807} C_VEL
LIN {X 0,Y 587.179,Z 482.431,A -85,B 0,C 180,E1 -1355.495,E2 -1355.495} C_VEL
LIN {X 0,Y 587.189,Z 479.661,A -85,B 0,C 180,E1 -1356.574,E2 -1356.574} C_VEL
LIN {X 0,Y 587.187,Z 476.137,A -85,B 0,C 180,E1 -1357.566,E2 -1357.566} C_VEL
LIN {X 0,Y 587.214,Z 471.323,A -85,B 0,C 180,E1 -1358.604,E2 -1358.604} C_VEL
LIN {X 0,Y 587.248,Z 465.261,A -85,B 0,C 180,E1 -1359.645,E2 -1359.645} C_VEL
LIN {X 0,Y 587.269,Z 457.698,A -85,B 0,C 180,E1 -1360.69,E2 -1360.69} C_VEL
LIN {X 0,Y 587.326,Z 448.19,A -85,B 0,C 180,E1 -1361.737,E2 -1361.737} C_VEL
LIN {X 0,Y 587.408,Z 438.334,A -85,B 0,C 180,E1 -1362.612,E2 -1362.612} C_VEL
LIN {X 0,Y 587.458,Z 427.25,A -85,B 0,C 180,E1 -1363.403,E2 -1363.403} C_VEL
LIN {X 0,Y 587.557,Z 415.675,A -85,B 0,C 180,E1 -1364.054,E2 -1364.054} C_VEL
LIN {X 0,Y 587.648,Z 403.273,A -85,B 0,C 180,E1 -1364.59,E2 -1364.59} C_VEL
LIN {X 0,Y 587.356,Z 398.323,A -85,B 0,C 180,E1 -1364.775,E2 -1364.775} C_VEL
LIN {X 0,Y 587.349,Z 398.317,A -85,B 0,C 180,E1 -1367.406,E2 -1367.406} C_VEL
LIN {X 0,Y 587.332,Z 398.328,A -85,B 0,C 180,E1 -1370.305,E2 -1370.305} C_VEL
LIN {X 0,Y 587.32,Z 398.32,A -85,B 0,C 180,E1 -1373.259,E2 -1373.259} C_VEL
LIN {X 0,Y 587.337,Z 398.318,A -85,B 0,C 180,E1 -1375.517,E2 -1375.517} C_VEL
LIN {X 0,Y 587.345,Z 398.32,A -85,B 0,C 180,E1 -1377.818,E2 -1377.818} C_VEL
LIN {X 0,Y 587.343,Z 398.323,A -85,B 0,C 180,E1 -1380.51,E2 -1380.51} C_VEL
LIN {X 0,Y 587.338,Z 398.318,A -85,B 0,C 180,E1 -1383.397,E2 -1383.397} C_VEL
LIN {X 0,Y 587.305,Z 398.327,A -85,B 0,C 180,E1 -1385.899,E2 -1385.899} C_VEL
LIN {X 0,Y 587.336,Z 398.323,A -85,B 0,C 180,E1 -1388.479,E2 -1388.479} C_VEL
LIN {X 0,Y 587.34,Z 398.317,A -85,B 0,C 180,E1 -1391.157,E2 -1391.157} C_VEL
LIN {X 0,Y 587.333,Z 398.328,A -85,B 0,C 180,E1 -1394.113,E2 -1394.113} C_VEL
LIN {X 0,Y 587.326,Z 398.319,A -85,B 0,C 180,E1 -1396.994,E2 -1396.994} C_VEL
LIN {X 0,Y 587.316,Z 398.326,A -85,B 0,C 180,E1 -1399.745,E2 -1399.745} C_VEL
LIN {X 0,Y 587.349,Z 398.32,A -85,B 0,C 180,E1 -1402.392,E2 -1402.392} C_VEL
LIN {X 0,Y 587.364,Z 398.322,A -85,B 0,C 180,E1 -1405.78,E2 -1405.78} C_VEL
LIN {X 0,Y 587.345,Z 398.322,A -85,B 0,C 180,E1 -1408.231,E2 -1408.231} C_VEL
LIN {X 0,Y 587.354,Z 398.316,A -85,B 0,C 180,E1 -1410.867,E2 -1410.867} C_VEL
LIN {X 0,Y 587.363,Z 398.325,A -85,B 0,C 180,E1 -1413.819,E2 -1413.819} C_VEL
LIN {X 0,Y 587.332,Z 398.326,A -85,B 0,C 180,E1 -1415.993,E2 -1415.993} C_VEL
LIN {X 0,Y 587.328,Z 398.322,A -85,B 0,C 180,E1 -1418.226,E2 -1418.226} C_VEL
LIN {X 0,Y 587.352,Z 398.318,A -85,B 0,C 180,E1 -1421.151,E2 -1421.151} C_VEL
LIN {X 0,Y 587.323,Z 398.325,A -85,B 0,C 180,E1 -1424.025,E2 -1424.025} C_VEL
LIN {X 0,Y 587.361,Z 398.318,A -85,B 0,C 180,E1 -1426.154,E2 -1426.154} C_VEL
LIN {X 0,Y 587.366,Z 398.32,A -85,B 0,C 180,E1 -1429.312,E2 -1429.312} C_VEL
LIN {X 0,Y 587.625,Z 404.188,A -85,B 0,C 180,E1 -1429.534,E2 -1429.534} C_VEL
LIN {X 0,Y 587.6,Z 416.93,A -85,B 0,C 180,E1 -1430.1,E2 -1430.1} C_VEL
LIN {X 0,Y 587.47,Z 427.513,A -85,B 0,C 180,E1 -1430.706,E2 -1430.706} C_VEL
LIN {X 0,Y 587.417,Z 437.315,A -85,B 0,C 180,E1 -1431.399,E2 -1431.399} C_VEL
LIN {X 0,Y 587.335,Z 447.286,A -85,B 0,C 180,E1 -1432.263,E2 -1432.263} C_VEL
LIN {X 0,Y 587.286,Z 455.418,A -85,B 0,C 180,E1 -1433.127,E2 -1433.127} C_VEL
LIN {X 0,Y 587.254,Z 463.386,A -85,B 0,C 180,E1 -1434.161,E2 -1434.161} C_VEL
LIN {X 0,Y 587.186,Z 469.774,A -85,B 0,C 180,E1 -1435.194,E2 -1435.194} C_VEL
LIN {X 0,Y 587.213,Z 474.875,A -85,B 0,C 180,E1 -1436.226,E2 -1436.226} C_VEL
LIN {X 0,Y 587.145,Z 478.833,A -85,B 0,C 180,E1 -1437.256,E2 -1437.256} C_VEL
LIN {X 0,Y 587.148,Z 482.514,A -85,B 0,C 180,E1 -1438.628,E2 -1438.628} C_VEL
LIN {X 0,Y 587.14,Z 483.719,A -85,B 0,C 180,E1 -1439.314,E2 -1439.314} C_VEL
LIN {X 0,Y 587.139,Z 484.926,A -85,B 0,C 180,E1 -1440.686,E2 -1440.686} C_VEL
LIN {X 0,Y 587.147,Z 484.934,A -85,B 0,C 180,E1 -1441.372,E2 -1441.372} C_VEL
LIN {X 0,Y 587.128,Z 483.77,A -85,B 0,C 180,E1 -1442.744,E2 -1442.744} C_VEL
LIN {X 0,Y 587.183,Z 482.578,A -85,B 0,C 180,E1 -1443.431,E2 -1443.431} C_VEL
LIN {X 0,Y 587.137,Z 478.932,A -85,B 0,C 180,E1 -1444.806,E2 -1444.806} C_VEL
LIN {X 0,Y 587.208,Z 474.99,A -85,B 0,C 180,E1 -1445.839,E2 -1445.839} C_VEL
LIN {X 0,Y 587.212,Z 469.896,A -85,B 0,C 180,E1 -1446.874,E2 -1446.874} C_VEL
LIN {X 0,Y 587.226,Z 463.507,A -85,B 0,C 180,E1 -1447.911,E2 -1447.911} C_VEL
LIN {X 0,Y 587.313,Z 455.534,A -85,B 0,C 180,E1 -1448.949,E2 -1448.949} C_VEL
LIN {X 0,Y 587.353,Z 447.377,A -85,B 0,C 180,E1 -1449.817,E2 -1449.817} C_VEL
LIN {X 0,Y 587.428,Z 437.369,A -85,B 0,C 180,E1 -1450.687,E2 -1450.687} C_VEL
LIN {X 0,Y 587.464,Z 427.516,A -85,B 0,C 180,E1 -1451.384,E2 -1451.384} C_VEL
LIN {X 0,Y 587.564,Z 416.853,A -85,B 0,C 180,E1 -1451.995,E2 -1451.995} C_VEL
LIN {X 0,Y 587.62,Z 403.985,A -85,B 0,C 180,E1 -1452.564,E2 -1452.564} C_VEL
LIN {X 0,Y 587.367,Z 398.321,A -85,B 0,C 180,E1 -1452.767,E2 -1452.767} C_VEL
LIN {X 0,Y 587.338,Z 398.324,A -85,B 0,C 180,E1 -1455.263,E2 -1455.263} C_VEL
LIN {X 0,Y 587.348,Z 398.327,A -85,B 0,C 180,E1 -1457.406,E2 -1457.406} C_VEL
LIN {X 0,Y 587.333,Z 398.329,A -85,B 0,C 180,E1 -1460.305,E2 -1460.305} C_VEL
LIN {X 0,Y 587.317,Z 398.328,A -85,B 0,C 180,E1 -1463.259,E2 -1463.259} C_VEL
LIN {X 0,Y 587.341,Z 398.325,A -85,B 0,C 180,E1 -1465.516,E2 -1465.516} C_VEL
LIN {X 0,Y 587.352,Z 398.321,A -85,B 0,C 180,E1 -1467.818,E2 -1467.818} C_VEL
LIN {X 0,Y 587.34,Z 398.323,A -85,B 0,C 180,E1 -1470.51,E2 -1470.51} C_VEL
LIN {X 0,Y 587.339,Z 398.323,A -85,B 0,C 180,E1 -1473.396,E2 -1473.396} C_VEL
LIN {X 0,Y 587.295,Z 398.33,A -85,B 0,C 180,E1 -1475.9,E2 -1475.9} C_VEL
LIN {X 0,Y 587.326,Z 398.328,A -85,B 0,C 180,E1 -1478.48,E2 -1478.48} C_VEL
LIN {X 0,Y 587.339,Z 398.327,A -85,B 0,C 180,E1 -1481.157,E2 -1481.157} C_VEL
LIN {X 0,Y 587.339,Z 398.326,A -85,B 0,C 180,E1 -1484.114,E2 -1484.114} C_VEL
LIN {X 0,Y 587.317,Z 398.328,A -85,B 0,C 180,E1 -1486.993,E2 -1486.993} C_VEL
LIN {X 0,Y 587.322,Z 398.328,A -85,B 0,C 180,E1 -1489.746,E2 -1489.746} C_VEL
LIN {X 0,Y 587.347,Z 398.327,A -85,B 0,C 180,E1 -1492.392,E2 -1492.392} C_VEL
LIN {X 0,Y 587.395,Z 398.481,A -85,B 0,C 180,E1 -1493.789,E2 -1493.789} C_VEL
LIN {X 0,Y 587.87,Z 402.816,A -85,B 0,C 180,E1 -1494.69,E2 -1494.69} C_VEL
LIN {X 0,Y 587.832,Z 420.233,A -85,B 0,C 180,E1 -1498.088,E2 -1498.088} C_VEL
LIN {X 0,Y 587.908,Z 434.544,A -85,B 0,C 180,E1 -1500.77,E2 -1500.77} C_VEL
LIN {X 0,Y 587.798,Z 447.756,A -85,B 0,C 180,E1 -1503.361,E2 -1503.361} C_VEL
LIN {X 0,Y 587.698,Z 461.449,A -85,B 0,C 180,E1 -1506.009,E2 -1506.009} C_VEL
LIN {X 0,Y 587.568,Z 475.146,A -85,B 0,C 180,E1 -1508.604,E2 -1508.604} C_VEL
LIN {X 0,Y 587.48,Z 490.796,A -85,B 0,C 180,E1 -1511.517,E2 -1511.517} C_VEL
LIN {X 0,Y 587.387,Z 506.447,A -85,B 0,C 180,E1 -1514.383,E2 -1514.383} C_VEL
LIN {X 0,Y 587.304,Z 522.098,A -85,B 0,C 180,E1 -1517.21,E2 -1517.21} C_VEL
LIN {X 0,Y 587.315,Z 525.155,A -85,B 0,C 180,E1 -1517.759,E2 -1517.759} C_VEL
LIN {X 0,Y 587.744,Z 530.936,A -85,B 0,C 180,E1 -1517.855,E2 -1517.855} C_VEL
LIN {X 0,Y 587.672,Z 544.211,A -85,B 0,C 180,E1 -1518.16,E2 -1518.16} C_VEL
LIN {X 0,Y 587.623,Z 556.659,A -85,B 0,C 180,E1 -1518.586,E2 -1518.586} C_VEL
LIN {X 0,Y 587.527,Z 568.628,A -85,B 0,C 180,E1 -1519.14,E2 -1519.14} C_VEL
LIN {X 0,Y 587.448,Z 580.198,A -85,B 0,C 180,E1 -1519.836,E2 -1519.836} C_VEL
LIN {X 0,Y 587.367,Z 590.595,A -85,B 0,C 180,E1 -1520.617,E2 -1520.617} C_VEL
LIN {X 0,Y 587.322,Z 599.11,A -85,B 0,C 180,E1 -1521.397,E2 -1521.397} C_VEL
LIN {X 0,Y 587.274,Z 606.959,A -85,B 0,C 180,E1 -1522.263,E2 -1522.263} C_VEL
LIN {X 0,Y 587.23,Z 613.468,A -85,B 0,C 180,E1 -1523.126,E2 -1523.126} C_VEL
LIN {X 0,Y 587.236,Z 619.865,A -85,B 0,C 180,E1 -1524.161,E2 -1524.161} C_VEL
LIN {X 0,Y 587.147,Z 624.949,A -85,B 0,C 180,E1 -1525.193,E2 -1525.193} C_VEL
LIN {X 0,Y 587.212,Z 628.895,A -85,B 0,C 180,E1 -1526.226,E2 -1526.226} C_VEL
LIN {X 0,Y 587.132,Z 631.808,A -85,B 0,C 180,E1 -1527.255,E2 -1527.255} C_VEL
LIN {X 0,Y 587.139,Z 633.2,A -85,B 0,C 180,E1 -1527.942,E2 -1527.942} C_VEL
LIN {X 0,Y 587.14,Z 634.784,A -85,B 0,C 180,E1 -1529.314,E2 -1529.314} C_VEL
LIN {X 0,Y 587.137,Z 635,A -85,B 0,C 180,E1 -1530,E2 -1530} C_VEL
LIN {X 0,Y 587.147,Z 634.185,A -85,B 0,C 180,E1 -1531.372,E2 -1531.372} C_VEL
LIN {X 0,Y 587.139,Z 633.202,A -85,B 0,C 180,E1 -1532.058,E2 -1532.058} C_VEL
LIN {X 0,Y 587.132,Z 631.81,A -85,B 0,C 180,E1 -1532.744,E2 -1532.744} C_VEL
LIN {X 0,Y 587.212,Z 628.896,A -85,B 0,C 180,E1 -1533.774,E2 -1533.774} C_VEL
LIN {X 0,Y 587.147,Z 624.95,A -85,B 0,C 180,E1 -1534.806,E2 -1534.806} C_VEL
LIN {X 0,Y 587.217,Z 618.878,A -85,B 0,C 180,E1 -1536.011,E2 -1536.011} C_VEL
LIN {X 0,Y 587.245,Z 612.237,A -85,B 0,C 180,E1 -1537.046,E2 -1537.046} C_VEL
LIN {X 0,Y 587.299,Z 603.991,A -85,B 0,C 180,E1 -1538.083,E2 -1538.083} C_VEL
LIN {X 0,Y 587.343,Z 595.539,A -85,B 0,C 180,E1 -1538.949,E2 -1538.949} C_VEL
LIN {X 0,Y 587.417,Z 585.096,A -85,B 0,C 180,E1 -1539.816,E2 -1539.816} C_VEL
LIN {X 0,Y 587.501,Z 574.76,A -85,B 0,C 180,E1 -1540.511,E2 -1540.511} C_VEL
LIN {X 0,Y 587.559,Z 562.833,A -85,B 0,C 180,E1 -1541.148,E2 -1541.148} C_VEL
LIN {X 0,Y 587.624,Z 550.609,A -85,B 0,C 180,E1 -1541.639,E2 -1541.639} C_VEL
LIN {X 0,Y 587.711,Z 537.441,A -85,B 0,C 180,E1 -1542.014,E2 -1542.014} C_VEL
LIN {X 0,Y 587.52,Z 526.608,A -85,B 0,C 180,E1 -1542.215,E2 -1542.215} C_VEL
LIN {X 0,Y 587.32,Z 525.035,A -85,B 0,C 180,E1 -1542.263,E2 -1542.263} C_VEL
LIN {X 0,Y 587.359,Z 510.362,A -85,B 0,C 180,E1 -1544.907,E2 -1544.907} C_VEL
LIN {X 0,Y 587.459,Z 494.71,A -85,B 0,C 180,E1 -1547.762,E2 -1547.762} C_VEL
LIN {X 0,Y 587.554,Z 479.059,A -85,B 0,C 180,E1 -1550.662,E2 -1550.662} C_VEL
LIN {X 0,Y 587.649,Z 465.364,A -85,B 0,C 180,E1 -1553.245,E2 -1553.245} C_VEL
LIN {X 0,Y 587.763,Z 451.669,A -85,B 0,C 180,E1 -1555.877,E2 -1555.877} C_VEL
LIN {X 0,Y 587.887,Z 437.974,A -85,B 0,C 180,E1 -1558.567,E2 -1558.567} C_VEL
LIN {X 0,Y 587.845,Z 424.354,A -85,B 0,C 180,E1 -1561.136,E2 -1561.136} C_VEL
LIN {X 0,Y 587.784,Z 409.522,A -85,B 0,C 180,E1 -1563.985,E2 -1563.985} C_VEL
LIN {X 0,Y 587.844,Z 401.373,A -85,B 0,C 180,E1 -1565.612,E2 -1565.612} C_VEL
LIN {X 0,Y 587.364,Z 398.325,A -85,B 0,C 180,E1 -1566.266,E2 -1566.266} C_VEL
LIN {X 0,Y 587.338,Z 398.326,A -85,B 0,C 180,E1 -1568.942,E2 -1568.942} C_VEL
LIN {X 0,Y 587.34,Z 398.325,A -85,B 0,C 180,E1 -1572.074,E2 -1572.074} C_VEL
LIN {X 0,Y 587.318,Z 398.328,A -85,B 0,C 180,E1 -1575.089,E2 -1575.089} C_VEL
LIN {X 0,Y 587.355,Z 398.326,A -85,B 0,C 180,E1 -1577.928,E2 -1577.928} C_VEL
LIN {X 0,Y 587.337,Z 398.327,A -85,B 0,C 180,E1 -1581.058,E2 -1581.058} C_VEL
LIN {X 0,Y 587.354,Z 398.325,A -85,B 0,C 180,E1 -1583.292,E2 -1583.292} C_VEL
LIN {X 0,Y 587.363,Z 398.323,A -85,B 0,C 180,E1 -1585.78,E2 -1585.78} C_VEL
LIN {X 0,Y 587.343,Z 398.325,A -85,B 0,C 180,E1 -1588.231,E2 -1588.231} C_VEL
LIN {X 0,Y 587.352,Z 398.326,A -85,B 0,C 180,E1 -1590.866,E2 -1590.866} C_VEL
LIN {X 0,Y 587.365,Z 398.322,A -85,B 0,C 180,E1 -1593.818,E2 -1593.818} C_VEL
LIN {X 0,Y 587.339,Z 398.325,A -85,B 0,C 180,E1 -1595.994,E2 -1595.994} C_VEL
LIN {X 0,Y 587.326,Z 398.327,A -85,B 0,C 180,E1 -1598.226,E2 -1598.226} C_VEL
LIN {X 0,Y 587.351,Z 398.323,A -85,B 0,C 180,E1 -1601.151,E2 -1601.151} C_VEL
LIN {X 0,Y 587.333,Z 398.328,A -85,B 0,C 180,E1 -1604.025,E2 -1604.025} C_VEL
LIN {X 0,Y 587.364,Z 398.325,A -85,B 0,C 180,E1 -1606.154,E2 -1606.154} C_VEL
LIN {X 0,Y 587.347,Z 398.324,A -85,B 0,C 180,E1 -1608.963,E2 -1608.963} C_VEL
LIN {X 0,Y 587.343,Z 398.326,A -85,B 0,C 180,E1 -1611.744,E2 -1611.744} C_VEL
LIN {X 0,Y 587.363,Z 398.323,A -85,B 0,C 180,E1 -1614.507,E2 -1614.507} C_VEL
LIN {X 0,Y 587.38,Z 398.321,A -85,B 0,C 180,E1 -1617.257,E2 -1617.257} C_VEL
LIN {X 0,Y 587.383,Z 398.321,A -85,B 0,C 180,E1 -1620,E2 -1620} C_VEL
LIN {X 0,Y 587.377,Z 398.32,A -85,B 0,C 180,E1 -1622.743,E2 -1622.743} C_VEL
LIN {X 0,Y 587.357,Z 398.324,A -85,B 0,C 180,E1 -1625.493,E2 -1625.493} C_VEL
LIN {X 0,Y 587.374,Z 398.321,A -85,B 0,C 180,E1 -1628.255,E2 -1628.255} C_VEL
LIN {X 0,Y 587.351,Z 398.326,A -85,B 0,C 180,E1 -1631.134,E2 -1631.134} C_VEL
LIN {X 0,Y 587.368,Z 398.324,A -85,B 0,C 180,E1 -1634.261,E2 -1634.261} C_VEL
LIN {X 0,Y 587.353,Z 398.325,A -85,B 0,C 180,E1 -1637.406,E2 -1637.406} C_VEL
LIN {X 0,Y 587.314,Z 398.327,A -85,B 0,C 180,E1 -1638.318,E2 -1638.318} C_VEL
LIN {X 0,Y 586.673,Z 398.409,A -85,B 0,C 180,E1 -1638.89,E2 -1638.89} C_VEL
LIN {X 0,Y 583.851,Z 398.762,A -85,B 0,C 180,E1 -1639.818,E2 -1639.818} C_VEL
LIN {X 0,Y 581.441,Z 399.062,A -85,B 0,C 180,E1 -1640.565,E2 -1640.565} C_VEL
LIN {X 0,Y 580.387,Z 399.192,A -85,B 0,C 180,E1 -1641.142,E2 -1641.142} C_VEL
LIN {X 0,Y 580.292,Z 399.203,A -85,B 0,C 180,E1 -1641.337,E2 -1641.337} C_VEL
LIN {X 0,Y 580.305,Z 399.202,A -85,B 0,C 180,E1 -1644.316,E2 -1644.316} C_VEL
LIN {X 0,Y 580.28,Z 399.204,A -85,B 0,C 180,E1 -1646.624,E2 -1646.624} C_VEL
LIN {X 0,Y 580.305,Z 399.202,A -85,B 0,C 180,E1 -1649.31,E2 -1649.31} C_VEL
LIN {X 0,Y 580.303,Z 399.202,A -85,B 0,C 180,E1 -1652.201,E2 -1652.201} C_VEL
LIN {X 0,Y 580.295,Z 399.204,A -85,B 0,C 180,E1 -1654.696,E2 -1654.696} C_VEL
LIN {X 0,Y 580.304,Z 399.202,A -85,B 0,C 180,E1 -1657.268,E2 -1657.268} C_VEL
LIN {X 0,Y 580.293,Z 399.206,A -85,B 0,C 180,E1 -1660.271,E2 -1660.271} C_VEL
LIN {X 0,Y 580.285,Z 399.204,A -85,B 0,C 180,E1 -1662.706,E2 -1662.706} C_VEL
LIN {X 0,Y 580.278,Z 399.207,A -85,B 0,C 180,E1 -1665.609,E2 -1665.609} C_VEL
LIN {X 0,Y 580.318,Z 399.2,A -85,B 0,C 180,E1 -1668.235,E2 -1668.235} C_VEL
LIN {X 0,Y 580.293,Z 399.204,A -85,B 0,C 180,E1 -1670.966,E2 -1670.966} C_VEL
LIN {X 0,Y 580.279,Z 399.205,A -85,B 0,C 180,E1 -1673.597,E2 -1673.597} C_VEL
LIN {X 0,Y 580.325,Z 399.199,A -85,B 0,C 180,E1 -1676.146,E2 -1676.146} C_VEL
LIN {X 0,Y 580.296,Z 399.205,A -85,B 0,C 180,E1 -1678.616,E2 -1678.616} C_VEL
LIN {X 0,Y 580.297,Z 399.204,A -85,B 0,C 180,E1 -1681.024,E2 -1681.024} C_VEL
LIN {X 0,Y 580.295,Z 399.203,A -85,B 0,C 180,E1 -1683.666,E2 -1683.666} C_VEL
LIN {X 0,Y 580.305,Z 399.201,A -85,B 0,C 180,E1 -1685.684,E2 -1685.684} C_VEL
LIN {X 0,Y 580.278,Z 399.205,A -85,B 0,C 180,E1 -1687.948,E2 -1687.948} C_VEL
LIN {X 0,Y 580.305,Z 399.202,A -85,B 0,C 180,E1 -1690.914,E2 -1690.914} C_VEL
LIN {X 0,Y 580.309,Z 399.201,A -85,B 0,C 180,E1 -1693.103,E2 -1693.103} C_VEL
LIN {X 0,Y 580.331,Z 399.201,A -85,B 0,C 180,E1 -1695.983,E2 -1695.983} C_VEL
LIN {X 0,Y 580.311,Z 399.201,A -85,B 0,C 180,E1 -1698.827,E2 -1698.827} C_VEL
LIN {X 0,Y 580.293,Z 399.204,A -85,B 0,C 180,E1 -1701.205,E2 -1701.205} C_VEL
LIN {X 0,Y 580.689,Z 402.766,A -85,B 0,C 180,E1 -1701.343,E2 -1701.343} C_VEL
LIN {X 0,Y 580.629,Z 414.11,A -85,B 0,C 180,E1 -1701.824,E2 -1701.824} C_VEL
LIN {X 0,Y 580.506,Z 425.233,A -85,B 0,C 180,E1 -1702.435,E2 -1702.435} C_VEL
LIN {X 0,Y 580.4,Z 436.103,A -85,B 0,C 180,E1 -1703.186,E2 -1703.186} C_VEL
LIN {X 0,Y 580.279,Z 444.772,A -85,B 0,C 180,E1 -1703.917,E2 -1703.917} C_VEL
LIN {X 0,Y 580.273,Z 453.291,A -85,B 0,C 180,E1 -1704.788,E2 -1704.788} C_VEL
LIN {X 0,Y 580.22,Z 461.672,A -85,B 0,C 180,E1 -1705.832,E2 -1705.832} C_VEL
LIN {X 0,Y 580.194,Z 468.392,A -85,B 0,C 180,E1 -1706.875,E2 -1706.875} C_VEL
LIN {X 0,Y 580.071,Z 473.772,A -85,B 0,C 180,E1 -1707.917,E2 -1707.917} C_VEL
LIN {X 0,Y 580.087,Z 477.979,A -85,B 0,C 180,E1 -1708.959,E2 -1708.959} C_VEL
LIN {X 0,Y 580.041,Z 481.139,A -85,B 0,C 180,E1 -1710,E2 -1710} C_VEL
LIN {X 0,Y 580.04,Z 482.697,A -85,B 0,C 180,E1 -1710.694,E2 -1710.694} C_VEL
LIN {X 0,Y 580.038,Z 484.606,A -85,B 0,C 180,E1 -1712.083,E2 -1712.083} C_VEL
LIN {X 0,Y 580.107,Z 484.911,A -85,B 0,C 180,E1 -1713.473,E2 -1713.473} C_VEL
LIN {X 0,Y 580.087,Z 484.478,A -85,B 0,C 180,E1 -1714.169,E2 -1714.169} C_VEL
LIN {X 0,Y 580.031,Z 483.62,A -85,B 0,C 180,E1 -1714.866,E2 -1714.866} C_VEL
LIN {X 0,Y 580.099,Z 482.352,A -85,B 0,C 180,E1 -1715.562,E2 -1715.562} C_VEL
LIN {X 0,Y 580.1,Z 479.831,A -85,B 0,C 180,E1 -1716.562,E2 -1716.562} C_VEL
LIN {X 0,Y 580.107,Z 475.986,A -85,B 0,C 180,E1 -1717.658,E2 -1717.658} C_VEL
LIN {X 0,Y 580.117,Z 471.122,A -85,B 0,C 180,E1 -1718.71,E2 -1718.71} C_VEL
LIN {X 0,Y 580.196,Z 465.016,A -85,B 0,C 180,E1 -1719.764,E2 -1719.764} C_VEL
LIN {X 0,Y 580.219,Z 457.71,A -85,B 0,C 180,E1 -1720.782,E2 -1720.782} C_VEL
LIN {X 0,Y 580.283,Z 449.591,A -85,B 0,C 180,E1 -1721.705,E2 -1721.705} C_VEL
LIN {X 0,Y 580.374,Z 438.944,A -85,B 0,C 180,E1 -1722.679,E2 -1722.679} C_VEL
LIN {X 0,Y 580.462,Z 429.335,A -85,B 0,C 180,E1 -1723.389,E2 -1723.389} C_VEL
LIN {X 0,Y 580.523,Z 419.012,A -85,B 0,C 180,E1 -1724.012,E2 -1724.012} C_VEL
LIN {X 0,Y 580.661,Z 407.775,A -85,B 0,C 180,E1 -1724.552,E2 -1724.552} C_VEL
LIN {X 0,Y 580.682,Z 400.849,A -85,B 0,C 180,E1 -1724.814,E2 -1724.814} C_VEL
LIN {X 0,Y 580.329,Z 399.197,A -85,B 0,C 180,E1 -1724.89,E2 -1724.89} C_VEL
LIN {X 0,Y 580.295,Z 399.197,A -85,B 0,C 180,E1 -1727.625,E2 -1727.625} C_VEL
LIN {X 0,Y 580.292,Z 399.198,A -85,B 0,C 180,E1 -1729.823,E2 -1729.823} C_VEL
LIN {X 0,Y 580.277,Z 399.203,A -85,B 0,C 180,E1 -1732.053,E2 -1732.053} C_VEL
LIN {X 0,Y 580.311,Z 399.194,A -85,B 0,C 180,E1 -1735.08,E2 -1735.08} C_VEL
LIN {X 0,Y 580.301,Z 399.203,A -85,B 0,C 180,E1 -1738.186,E2 -1738.186} C_VEL
LIN {X 0,Y 580.29,Z 399.199,A -85,B 0,C 180,E1 -1740.695,E2 -1740.695} C_VEL
LIN {X 0,Y 580.307,Z 399.194,A -85,B 0,C 180,E1 -1743.316,E2 -1743.316} C_VEL
LIN {X 0,Y 580.27,Z 399.202,A -85,B 0,C 180,E1 -1745.759,E2 -1745.759} C_VEL
LIN {X 0,Y 580.294,Z 399.206,A -85,B 0,C 180,E1 -1748.146,E2 -1748.146} C_VEL
LIN {X 0,Y 580.302,Z 399.195,A -85,B 0,C 180,E1 -1750.843,E2 -1750.843} C_VEL
LIN {X 0,Y 580.284,Z 399.2,A -85,B 0,C 180,E1 -1753.658,E2 -1753.658} C_VEL
LIN {X 0,Y 580.291,Z 399.198,A -85,B 0,C 180,E1 -1756.608,E2 -1756.608} C_VEL
LIN {X 0,Y 580.302,Z 399.194,A -85,B 0,C 180,E1 -1759.156,E2 -1759.156} C_VEL
LIN {X 0,Y 580.295,Z 399.205,A -85,B 0,C 180,E1 -1761.927,E2 -1761.927} C_VEL
LIN {X 0,Y 580.255,Z 399.203,A -85,B 0,C 180,E1 -1764.453,E2 -1764.453} C_VEL
LIN {X 0,Y 580.295,Z 399.195,A -85,B 0,C 180,E1 -1766.975,E2 -1766.975} C_VEL
LIN {X 0,Y 580.3,Z 399.197,A -85,B 0,C 180,E1 -1769.425,E2 -1769.425} C_VEL
LIN {X 0,Y 580.297,Z 399.2,A -85,B 0,C 180,E1 -1772.142,E2 -1772.142} C_VEL
LIN {X 0,Y 580.31,Z 399.193,A -85,B 0,C 180,E1 -1774.92,E2 -1774.92} C_VEL
LIN {X 0,Y 580.278,Z 399.205,A -85,B 0,C 180,E1 -1777.947,E2 -1777.947} C_VEL
LIN {X 0,Y 580.302,Z 399.194,A -85,B 0,C 180,E1 -1780.913,E2 -1780.913} C_VEL
LIN {X 0,Y 580.275,Z 399.206,A -85,B 0,C 180,E1 -1783.825,E2 -1783.825} C_VEL
LIN {X 0,Y 580.329,Z 399.197,A -85,B 0,C 180,E1 -1785.983,E2 -1785.983} C_VEL
LIN {X 0,Y 580.311,Z 399.195,A -85,B 0,C 180,E1 -1788.827,E2 -1788.827} C_VEL
LIN {X 0,Y 580.329,Z 399.196,A -85,B 0,C 180,E1 -1789.209,E2 -1789.209} C_VEL
LIN {X 0,Y 580.689,Z 403.766,A -85,B 0,C 180,E1 -1789.378,E2 -1789.378} C_VEL
LIN {X 0,Y 580.601,Z 415.451,A -85,B 0,C 180,E1 -1789.891,E2 -1789.891} C_VEL
LIN {X 0,Y 580.467,Z 426.346,A -85,B 0,C 180,E1 -1790.505,E2 -1790.505} C_VEL
LIN {X 0,Y 580.379,Z 436.338,A -85,B 0,C 180,E1 -1791.206,E2 -1791.206} C_VEL
LIN {X 0,Y 580.339,Z 445.573,A -85,B 0,C 180,E1 -1791.994,E2 -1791.994} C_VEL
LIN {X 0,Y 580.248,Z 454.042,A -85,B 0,C 180,E1 -1792.868,E2 -1792.868} C_VEL
LIN {X 0,Y 580.209,Z 462.265,A -85,B 0,C 180,E1 -1793.916,E2 -1793.916} C_VEL
LIN {X 0,Y 580.102,Z 467.879,A -85,B 0,C 180,E1 -1794.787,E2 -1794.787} C_VEL
LIN {X 0,Y 580.108,Z 473.36,A -85,B 0,C 180,E1 -1795.831,E2 -1795.831} C_VEL
LIN {X 0,Y 580.093,Z 477.656,A -85,B 0,C 180,E1 -1796.875,E2 -1796.875} C_VEL
LIN {X 0,Y 580.048,Z 480.898,A -85,B 0,C 180,E1 -1797.917,E2 -1797.917} C_VEL
LIN {X 0,Y 580.048,Z 482.542,A -85,B 0,C 180,E1 -1798.611,E2 -1798.611} C_VEL
LIN {X 0,Y 580.04,Z 483.738,A -85,B 0,C 180,E1 -1799.306,E2 -1799.306} C_VEL
LIN {X 0,Y 580.039,Z 484.93,A -85,B 0,C 180,E1 -1800.694,E2 -1800.694} C_VEL
LIN {X 0,Y 580.047,Z 484.931,A -85,B 0,C 180,E1 -1801.388,E2 -1801.388} C_VEL
LIN {X 0,Y 580.04,Z 483.748,A -85,B 0,C 180,E1 -1802.778,E2 -1802.778} C_VEL
LIN {X 0,Y 580.109,Z 482.554,A -85,B 0,C 180,E1 -1803.473,E2 -1803.473} C_VEL
LIN {X 0,Y 580.041,Z 478.881,A -85,B 0,C 180,E1 -1804.865,E2 -1804.865} C_VEL
LIN {X 0,Y 580.118,Z 474.925,A -85,B 0,C 180,E1 -1805.91,E2 -1805.91} C_VEL
LIN {X 0,Y 580.143,Z 469.817,A -85,B 0,C 180,E1 -1806.958,E2 -1806.958} C_VEL
LIN {X 0,Y 580.172,Z 463.413,A -85,B 0,C 180,E1 -1808.008,E2 -1808.008} C_VEL
LIN {X 0,Y 580.252,Z 455.426,A -85,B 0,C 180,E1 -1809.059,E2 -1809.059} C_VEL
LIN {X 0,Y 580.307,Z 447.249,A -85,B 0,C 180,E1 -1809.938,E2 -1809.938} C_VEL
LIN {X 0,Y 580.413,Z 437.355,A -85,B 0,C 180,E1 -1810.805,E2 -1810.805} C_VEL
LIN {X 0,Y 580.479,Z 427.301,A -85,B 0,C 180,E1 -1811.523,E2 -1811.523} C_VEL
LIN {X 0,Y 580.591,Z 416.596,A -85,B 0,C 180,E1 -1812.141,E2 -1812.141} C_VEL
LIN {X 0,Y 580.686,Z 403.659,A -85,B 0,C 180,E1 -1812.716,E2 -1812.716} C_VEL
LIN {X 0,Y 580.343,Z 399.471,A -85,B 0,C 180,E1 -1812.868,E2 -1812.868} C_VEL
LIN {X 0,Y 580.306,Z 399.201,A -85,B 0,C 180,E1 -1812.903,E2 -1812.903} C_VEL
LIN {X 0,Y 580.303,Z 399.2,A -85,B 0,C 180,E1 -1815.453,E2 -1815.453} C_VEL
LIN {X 0,Y 580.292,Z 399.205,A -85,B 0,C 180,E1 -1817.625,E2 -1817.625} C_VEL
LIN {X 0,Y 580.309,Z 399.201,A -85,B 0,C 180,E1 -1819.822,E2 -1819.822} C_VEL
LIN {X 0,Y 580.295,Z 399.204,A -85,B 0,C 180,E1 -1822.802,E2 -1822.802} C_VEL
LIN {X 0,Y 580.312,Z 399.199,A -85,B 0,C 180,E1 -1825.08,E2 -1825.08} C_VEL
LIN {X 0,Y 580.305,Z 399.2,A -85,B 0,C 180,E1 -1828.185,E2 -1828.185} C_VEL
LIN {X 0,Y 580.288,Z 399.202,A -85,B 0,C 180,E1 -1830.694,E2 -1830.694} C_VEL
LIN {X 0,Y 580.308,Z 399.199,A -85,B 0,C 180,E1 -1833.316,E2 -1833.316} C_VEL
LIN {X 0,Y 580.25,Z 399.209,A -85,B 0,C 180,E1 -1835.756,E2 -1835.756} C_VEL
LIN {X 0,Y 580.289,Z 399.204,A -85,B 0,C 180,E1 -1838.146,E2 -1838.146} C_VEL
LIN {X 0,Y 580.301,Z 399.202,A -85,B 0,C 180,E1 -1840.843,E2 -1840.843} C_VEL
LIN {X 0,Y 580.293,Z 399.203,A -85,B 0,C 180,E1 -1843.657,E2 -1843.657} C_VEL
LIN {X 0,Y 580.278,Z 399.206,A -85,B 0,C 180,E1 -1846.609,E2 -1846.609} C_VEL
LIN {X 0,Y 580.302,Z 399.202,A -85,B 0,C 180,E1 -1849.156,E2 -1849.156} C_VEL
LIN {X 0,Y 580.293,Z 399.203,A -85,B 0,C 180,E1 -1851.927,E2 -1851.927} C_VEL
LIN {X 0,Y 580.34,Z 399.298,A -85,B 0,C 180,E1 -1853.577,E2 -1853.577} C_VEL
LIN {X 0,Y 580.923,Z 403.633,A -85,B 0,C 180,E1 -1854.5,E2 -1854.5} C_VEL
LIN {X 0,Y 580.849,Z 417.304,A -85,B 0,C 180,E1 -1857.217,E2 -1857.217} C_VEL
LIN {X 0,Y 580.944,Z 432.14,A -85,B 0,C 180,E1 -1860.064,E2 -1860.064} C_VEL
LIN {X 0,Y 580.935,Z 445.798,A -85,B 0,C 180,E1 -1862.631,E2 -1862.631} C_VEL
LIN {X 0,Y 580.766,Z 460.079,A -85,B 0,C 180,E1 -1865.438,E2 -1865.438} C_VEL
LIN {X 0,Y 580.625,Z 473.188,A -85,B 0,C 180,E1 -1867.961,E2 -1867.961} C_VEL
LIN {X 0,Y 580.508,Z 488.839,A -85,B 0,C 180,E1 -1870.92,E2 -1870.92} C_VEL
LIN {X 0,Y 580.348,Z 504.491,A -85,B 0,C 180,E1 -1873.827,E2 -1873.827} C_VEL
LIN {X 0,Y 580.302,Z 518.186,A -85,B 0,C 180,E1 -1876.34,E2 -1876.34} C_VEL
LIN {X 0,Y 580.271,Z 525.155,A -85,B 0,C 180,E1 -1877.608,E2 -1877.608} C_VEL
LIN {X 0,Y 580.806,Z 530.936,A -85,B 0,C 180,E1 -1877.708,E2 -1877.708} C_VEL
LIN {X 0,Y 580.745,Z 544.212,A -85,B 0,C 180,E1 -1878.017,E2 -1878.017} C_VEL
LIN {X 0,Y 580.666,Z 556.367,A -85,B 0,C 180,E1 -1878.436,E2 -1878.436} C_VEL
LIN {X 0,Y 580.55,Z 568.627,A -85,B 0,C 180,E1 -1879.008,E2 -1879.008} C_VEL
LIN {X 0,Y 580.422,Z 580.199,A -85,B 0,C 180,E1 -1879.712,E2 -1879.712} C_VEL
LIN {X 0,Y 580.346,Z 590.596,A -85,B 0,C 180,E1 -1880.503,E2 -1880.503} C_VEL
LIN {X 0,Y 580.271,Z 599.11,A -85,B 0,C 180,E1 -1881.292,E2 -1881.292} C_VEL
LIN {X 0,Y 580.222,Z 606.959,A -85,B 0,C 180,E1 -1882.168,E2 -1882.168} C_VEL
LIN {X 0,Y 580.154,Z 614.649,A -85,B 0,C 180,E1 -1883.221,E2 -1883.221} C_VEL
LIN {X 0,Y 580.139,Z 621.679,A -85,B 0,C 180,E1 -1884.438,E2 -1884.438} C_VEL
LIN {X 0,Y 580.108,Z 626.371,A -85,B 0,C 180,E1 -1885.483,E2 -1885.483} C_VEL
LIN {X 0,Y 580.123,Z 629.956,A -85,B 0,C 180,E1 -1886.527,E2 -1886.527} C_VEL
LIN {X 0,Y 580.043,Z 631.808,A -85,B 0,C 180,E1 -1887.222,E2 -1887.222} C_VEL
LIN {X 0,Y 580.038,Z 633.2,A -85,B 0,C 180,E1 -1887.917,E2 -1887.917} C_VEL
LIN {X 0,Y 580.04,Z 634.784,A -85,B 0,C 180,E1 -1889.306,E2 -1889.306} C_VEL
LIN {X 0,Y 580.037,Z 635,A -85,B 0,C 180,E1 -1890,E2 -1890} C_VEL
LIN {X 0,Y 580.047,Z 634.186,A -85,B 0,C 180,E1 -1891.388,E2 -1891.388} C_VEL
LIN {X 0,Y 580.038,Z 633.201,A -85,B 0,C 180,E1 -1892.083,E2 -1892.083} C_VEL
LIN {X 0,Y 580.043,Z 631.81,A -85,B 0,C 180,E1 -1892.778,E2 -1892.778} C_VEL
LIN {X 0,Y 580.109,Z 628.896,A -85,B 0,C 180,E1 -1893.82,E2 -1893.82} C_VEL
LIN {X 0,Y 580.054,Z 624.95,A -85,B 0,C 180,E1 -1894.865,E2 -1894.865} C_VEL
LIN {X 0,Y 580.139,Z 618.878,A -85,B 0,C 180,E1 -1896.085,E2 -1896.085} C_VEL
LIN {X 0,Y 580.184,Z 612.238,A -85,B 0,C 180,E1 -1897.132,E2 -1897.132} C_VEL
LIN {X 0,Y 580.25,Z 603.991,A -85,B 0,C 180,E1 -1898.182,E2 -1898.182} C_VEL
LIN {X 0,Y 580.308,Z 595.539,A -85,B 0,C 180,E1 -1899.058,E2 -1899.058} C_VEL
LIN {X 0,Y 580.417,Z 585.097,A -85,B 0,C 180,E1 -1899.936,E2 -1899.936} C_VEL
LIN {X 0,Y 580.506,Z 574.759,A -85,B 0,C 180,E1 -1900.639,E2 -1900.639} C_VEL
LIN {X 0,Y 580.595,Z 563.262,A -85,B 0,C 180,E1 -1901.263,E2 -1901.263} C_VEL
LIN {X 0,Y 580.659,Z 550.474,A -85,B 0,C 180,E1 -1901.785,E2 -1901.785} C_VEL
LIN {X 0,Y 580.785,Z 537.44,A -85,B 0,C 180,E1 -1902.159,E2 -1902.159} C_VEL
LIN {X 0,Y 580.633,Z 527.55,A -85,B 0,C 180,E1 -1902.348,E2 -1902.348} C_VEL
LIN {X 0,Y 580.255,Z 525.035,A -85,B 0,C 180,E1 -1902.415,E2 -1902.415} C_VEL
LIN {X 0,Y 580.34,Z 510.362,A -85,B 0,C 180,E1 -1905.092,E2 -1905.092} C_VEL
LIN {X 0,Y 580.442,Z 494.71,A -85,B 0,C 180,E1 -1907.984,E2 -1907.984} C_VEL
LIN {X 0,Y 580.584,Z 479.223,A -85,B 0,C 180,E1 -1910.891,E2 -1910.891} C_VEL
LIN {X 0,Y 580.734,Z 463.407,A -85,B 0,C 180,E1 -1913.917,E2 -1913.917} C_VEL
LIN {X 0,Y 580.883,Z 449.712,A -85,B 0,C 180,E1 -1916.593,E2 -1916.593} C_VEL
LIN {X 0,Y 580.907,Z 439.551,A -85,B 0,C 180,E1 -1918.547,E2 -1918.547} C_VEL
LIN {X 0,Y 580.898,Z 426.434,A -85,B 0,C 180,E1 -1921.031,E2 -1921.031} C_VEL
LIN {X 0,Y 580.88,Z 411.023,A -85,B 0,C 180,E1 -1924.025,E2 -1924.025} C_VEL
LIN {X 0,Y 580.843,Z 402.077,A -85,B 0,C 180,E1 -1925.838,E2 -1925.838} C_VEL
LIN {X 0,Y 580.329,Z 399.2,A -85,B 0,C 180,E1 -1926.495,E2 -1926.495} C_VEL
LIN {X 0,Y 580.312,Z 399.203,A -85,B 0,C 180,E1 -1929.187,E2 -1929.187} C_VEL
LIN {X 0,Y 580.292,Z 399.204,A -85,B 0,C 180,E1 -1931.768,E2 -1931.768} C_VEL
LIN {X 0,Y 580.265,Z 399.209,A -85,B 0,C 180,E1 -1934.626,E2 -1934.626} C_VEL
LIN {X 0,Y 580.284,Z 399.204,A -85,B 0,C 180,E1 -1937.294,E2 -1937.294} C_VEL
LIN {X 0,Y 580.297,Z 399.205,A -85,B 0,C 180,E1 -1940.067,E2 -1940.067} C_VEL
LIN {X 0,Y 580.303,Z 399.202,A -85,B 0,C 180,E1 -1943.065,E2 -1943.065} C_VEL
LIN {X 0,Y 580.317,Z 399.2,A -85,B 0,C 180,E1 -1946.145,E2 -1946.145} C_VEL
LIN {X 0,Y 580.279,Z 399.206,A -85,B 0,C 180,E1 -1948.615,E2 -1948.615} C_VEL
LIN {X 0,Y 580.296,Z 399.204,A -85,B 0,C 180,E1 -1951.024,E2 -1951.024} C_VEL
LIN {X 0,Y 580.331,Z 399.198,A -85,B 0,C 180,E1 -1953.658,E2 -1953.658} C_VEL
LIN {X 0,Y 580.282,Z 399.206,A -85,B 0,C 180,E1 -1956.442,E2 -1956.442} C_VEL
LIN {X 0,Y 580.276,Z 399.206,A -85,B 0,C 180,E1 -1959.437,E2 -1959.437} C_VEL
LIN {X 0,Y 580.269,Z 399.207,A -85,B 0,C 180,E1 -1961.645,E2 -1961.645} C_VEL
LIN {X 0,Y 580.286,Z 399.205,A -85,B 0,C 180,E1 -1963.826,E2 -1963.826} C_VEL
LIN {X 0,Y 580.33,Z 399.2,A -85,B 0,C 180,E1 -1965.983,E2 -1965.983} C_VEL
LIN {X 0,Y 580.307,Z 399.201,A -85,B 0,C 180,E1 -1968.827,E2 -1968.827} C_VEL
LIN {X 0,Y 580.312,Z 399.203,A -85,B 0,C 180,E1 -1971.644,E2 -1971.644} C_VEL
LIN {X 0,Y 580.286,Z 399.207,A -85,B 0,C 180,E1 -1973.742,E2 -1973.742} C_VEL
LIN {X 0,Y 580.277,Z 399.207,A -85,B 0,C 180,E1 -1975.833,E2 -1975.833} C_VEL
LIN {X 0,Y 580.347,Z 399.198,A -85,B 0,C 180,E1 -1977.918,E2 -1977.918} C_VEL
LIN {X 0,Y 580.367,Z 399.193,A -85,B 0,C 180,E1 -1980.694,E2 -1980.694} C_VEL
LIN {X 0,Y 580.283,Z 399.207,A -85,B 0,C 180,E1 -1983.472,E2 -1983.472} C_VEL
LIN {X 0,Y 580.323,Z 399.201,A -85,B 0,C 180,E1 -1985.56,E2 -1985.56} C_VEL
LIN {X 0,Y 580.338,Z 399.197,A -85,B 0,C 180,E1 -1988.356,E2 -1988.356} C_VEL
LIN {X 0,Y 580.303,Z 399.203,A -85,B 0,C 180,E1 -1991.191,E2 -1991.191} C_VEL
LIN {X 0,Y 580.33,Z 399.199,A -85,B 0,C 180,E1 -1994.017,E2 -1994.017} C_VEL
LIN {X 0,Y 580.315,Z 399.199,A -85,B 0,C 180,E1 -1996.914,E2 -1996.914} C_VEL
LIN {X 0,Y 580.31,Z 399.203,A -85,B 0,C 180,E1 -1999.822,E2 -1999.822} C_VEL
LIN {X 0,Y 580.292,Z 399.203,A -85,B 0,C 180,E1 -2001.337,E2 -2001.337} C_VEL
LIN {X 0,Y 579.593,Z 399.293,A -85,B 0,C 180,E1 -2001.916,E2 -2001.916} C_VEL
LIN {X 0,Y 576.715,Z 399.651,A -85,B 0,C 180,E1 -2002.856,E2 -2002.856} C_VEL
LIN {X 0,Y 574.32,Z 399.947,A -85,B 0,C 180,E1 -2003.612,E2 -2003.612} C_VEL
LIN {X 0,Y 573.321,Z 400.073,A -85,B 0,C 180,E1 -2004.196,E2 -2004.196} C_VEL
LIN {X 0,Y 573.254,Z 400.078,A -85,B 0,C 180,E1 -2004.393,E2 -2004.393} C_VEL
LIN {X 0,Y 573.254,Z 400.08,A -85,B 0,C 180,E1 -2006.976,E2 -2006.976} C_VEL
LIN {X 0,Y 573.25,Z 400.083,A -85,B 0,C 180,E1 -2009.489,E2 -2009.489} C_VEL
LIN {X 0,Y 573.258,Z 400.081,A -85,B 0,C 180,E1 -2012.645,E2 -2012.645} C_VEL
LIN {X 0,Y 573.259,Z 400.08,A -85,B 0,C 180,E1 -2015.185,E2 -2015.185} C_VEL
LIN {X 0,Y 573.24,Z 400.082,A -85,B 0,C 180,E1 -2017.808,E2 -2017.808} C_VEL
LIN {X 0,Y 573.247,Z 400.081,A -85,B 0,C 180,E1 -2020.525,E2 -2020.525} C_VEL
LIN {X 0,Y 573.251,Z 400.081,A -85,B 0,C 180,E1 -2023.358,E2 -2023.358} C_VEL
LIN {X 0,Y 573.256,Z 400.079,A -85,B 0,C 180,E1 -2026.33,E2 -2026.33} C_VEL
LIN {X 0,Y 573.263,Z 400.079,A -85,B 0,C 180,E1 -2029.476,E2 -2029.476} C_VEL
LIN {X 0,Y 573.239,Z 400.084,A -85,B 0,C 180,E1 -2032.193,E2 -2032.193} C_VEL
LIN {X 0,Y 573.256,Z 400.08,A -85,B 0,C 180,E1 -2035.226,E2 -2035.226} C_VEL
LIN {X 0,Y 573.261,Z 400.08,A -85,B 0,C 180,E1 -2037.771,E2 -2037.771} C_VEL
LIN {X 0,Y 573.273,Z 400.078,A -85,B 0,C 180,E1 -2040.635,E2 -2040.635} C_VEL
LIN {X 0,Y 573.24,Z 400.082,A -85,B 0,C 180,E1 -2043.508,E2 -2043.508} C_VEL
LIN {X 0,Y 573.236,Z 400.084,A -85,B 0,C 180,E1 -2046.135,E2 -2046.135} C_VEL
LIN {X 0,Y 573.256,Z 400.079,A -85,B 0,C 180,E1 -2049.174,E2 -2049.174} C_VEL
LIN {X 0,Y 573.236,Z 400.082,A -85,B 0,C 180,E1 -2051.412,E2 -2051.412} C_VEL
LIN {X 0,Y 573.248,Z 400.081,A -85,B 0,C 180,E1 -2053.622,E2 -2053.622} C_VEL
LIN {X 0,Y 573.278,Z 400.078,A -85,B 0,C 180,E1 -2055.807,E2 -2055.807} C_VEL
LIN {X 0,Y 573.269,Z 400.078,A -85,B 0,C 180,E1 -2058.745,E2 -2058.745} C_VEL
LIN {X 0,Y 573.279,Z 400.092,A -85,B 0,C 180,E1 -2061.096,E2 -2061.096} C_VEL
LIN {X 0,Y 573.713,Z 403.815,A -85,B 0,C 180,E1 -2061.236,E2 -2061.236} C_VEL
LIN {X 0,Y 573.615,Z 416.6,A -85,B 0,C 180,E1 -2061.812,E2 -2061.812} C_VEL
LIN {X 0,Y 573.481,Z 427.192,A -85,B 0,C 180,E1 -2062.43,E2 -2062.43} C_VEL
LIN {X 0,Y 573.382,Z 436.971,A -85,B 0,C 180,E1 -2063.135,E2 -2063.135} C_VEL
LIN {X 0,Y 573.235,Z 445.188,A -85,B 0,C 180,E1 -2063.842,E2 -2063.842} C_VEL
LIN {X 0,Y 573.229,Z 453.614,A -85,B 0,C 180,E1 -2064.724,E2 -2064.724} C_VEL
LIN {X 0,Y 573.145,Z 461.939,A -85,B 0,C 180,E1 -2065.781,E2 -2065.781} C_VEL
LIN {X 0,Y 573.104,Z 468.611,A -85,B 0,C 180,E1 -2066.837,E2 -2066.837} C_VEL
LIN {X 0,Y 572.978,Z 473.947,A -85,B 0,C 180,E1 -2067.891,E2 -2067.891} C_VEL
LIN {X 0,Y 573.01,Z 478.113,A -85,B 0,C 180,E1 -2068.946,E2 -2068.946} C_VEL
LIN {X 0,Y 572.942,Z 481.236,A -85,B 0,C 180,E1 -2070,E2 -2070} C_VEL
LIN {X 0,Y 572.941,Z 482.772,A -85,B 0,C 180,E1 -2070.703,E2 -2070.703} C_VEL
LIN {X 0,Y 572.938,Z 484.632,A -85,B 0,C 180,E1 -2072.109,E2 -2072.109} C_VEL
LIN {X 0,Y 573.006,Z 484.903,A -85,B 0,C 180,E1 -2073.516,E2 -2073.516} C_VEL
LIN {X 0,Y 573.007,Z 484.436,A -85,B 0,C 180,E1 -2074.22,E2 -2074.22} C_VEL
LIN {X 0,Y 572.94,Z 483.562,A -85,B 0,C 180,E1 -2074.926,E2 -2074.926} C_VEL
LIN {X 0,Y 572.975,Z 480.602,A -85,B 0,C 180,E1 -2076.338,E2 -2076.338} C_VEL
LIN {X 0,Y 573.006,Z 477.212,A -85,B 0,C 180,E1 -2077.4,E2 -2077.4} C_VEL
LIN {X 0,Y 573.053,Z 472.721,A -85,B 0,C 180,E1 -2078.463,E2 -2078.463} C_VEL
LIN {X 0,Y 573.062,Z 466.981,A -85,B 0,C 180,E1 -2079.53,E2 -2079.53} C_VEL
LIN {X 0,Y 573.103,Z 459.854,A -85,B 0,C 180,E1 -2080.6,E2 -2080.6} C_VEL
LIN {X 0,Y 573.234,Z 450.89,A -85,B 0,C 180,E1 -2081.671,E2 -2081.671} C_VEL
LIN {X 0,Y 573.281,Z 441.68,A -85,B 0,C 180,E1 -2082.568,E2 -2082.568} C_VEL
LIN {X 0,Y 573.407,Z 431.389,A -85,B 0,C 180,E1 -2083.376,E2 -2083.376} C_VEL
LIN {X 0,Y 573.521,Z 421.536,A -85,B 0,C 180,E1 -2084.006,E2 -2084.006} C_VEL
LIN {X 0,Y 573.65,Z 410.049,A -85,B 0,C 180,E1 -2084.595,E2 -2084.595} C_VEL
LIN {X 0,Y 573.747,Z 402.315,A -85,B 0,C 180,E1 -2084.906,E2 -2084.906} C_VEL
LIN {X 0,Y 573.294,Z 400.073,A -85,B 0,C 180,E1 -2085.009,E2 -2085.009} C_VEL
LIN {X 0,Y 573.247,Z 400.076,A -85,B 0,C 180,E1 -2087.849,E2 -2087.849} C_VEL
LIN {X 0,Y 573.247,Z 400.079,A -85,B 0,C 180,E1 -2090.077,E2 -2090.077} C_VEL
LIN {X 0,Y 573.24,Z 400.084,A -85,B 0,C 180,E1 -2092.338,E2 -2092.338} C_VEL
LIN {X 0,Y 573.259,Z 400.072,A -85,B 0,C 180,E1 -2095.41,E2 -2095.41} C_VEL
LIN {X 0,Y 573.241,Z 400.079,A -85,B 0,C 180,E1 -2098.565,E2 -2098.565} C_VEL
LIN {X 0,Y 573.231,Z 400.076,A -85,B 0,C 180,E1 -2100.993,E2 -2100.993} C_VEL
LIN {X 0,Y 573.268,Z 400.071,A -85,B 0,C 180,E1 -2103.524,E2 -2103.524} C_VEL
LIN {X 0,Y 573.245,Z 400.081,A -85,B 0,C 180,E1 -2106.05,E2 -2106.05} C_VEL
LIN {X 0,Y 573.249,Z 400.075,A -85,B 0,C 180,E1 -2108.701,E2 -2108.701} C_VEL
LIN {X 0,Y 573.235,Z 400.077,A -85,B 0,C 180,E1 -2111.593,E2 -2111.593} C_VEL
LIN {X 0,Y 573.241,Z 400.08,A -85,B 0,C 180,E1 -2114.333,E2 -2114.333} C_VEL
LIN {X 0,Y 573.249,Z 400.074,A -85,B 0,C 180,E1 -2117.358,E2 -2117.358} C_VEL
LIN {X 0,Y 573.243,Z 400.077,A -85,B 0,C 180,E1 -2120.392,E2 -2120.392} C_VEL
LIN {X 0,Y 573.257,Z 400.072,A -85,B 0,C 180,E1 -2123.078,E2 -2123.078} C_VEL
